C05463=1023.749,201.807,381.412,168.832,48.309,159.110
C05464=1023.754,202.056,381.388,168.836,48.304,159.109
C05465=1023.760,202.305,381.365,168.841,48.300,159.109
C05466=1023.765,202.553,381.340,168.844,48.295,159.109
C05467=1023.771,202.803,381.316,168.849,48.290,159.108
C05468=1023.776,203.051,381.291,168.853,48.285,159.108
C05469=1023.782,203.300,381.268,168.857,48.280,159.107
C05470=1023.805,204.331,381.167,169.270,48.380,159.187
C05471=1023.816,204.745,381.124,169.275,48.373,159.186
C05472=1023.827,205.160,381.081,169.281,48.366,159.186
C05473=1023.838,205.574,381.039,169.286,48.359,159.185
C05474=1023.849,205.988,380.996,169.292,48.352,159.184
C05475=1023.856,206.237,380.969,169.295,48.349,159.184
C05476=1023.862,206.486,380.944,169.298,48.344,159.184
C05477=1023.868,206.734,380.918,169.301,48.341,159.183
C05478=1023.874,206.982,380.892,169.305,48.336,159.183
C05479=1023.882,207.231,380.866,169.307,48.333,159.182
C05480=1023.888,207.480,380.841,169.311,48.329,159.182
C05481=1023.894,207.728,380.815,169.314,48.325,159.182
C05482=1023.900,207.976,380.789,169.318,48.321,159.181
C05483=1023.908,208.225,380.763,169.320,48.317,159.181
C05484=1023.913,208.474,380.737,169.324,48.313,159.180
C05485=1023.920,208.722,380.711,169.327,48.309,159.180
C05486=1023.926,208.972,380.685,169.331,48.305,159.180
C05487=1023.933,209.220,380.659,169.333,48.301,159.179
C05488=1023.939,209.468,380.633,169.337,48.297,159.179
C05489=1023.946,209.717,380.607,169.340,48.293,159.179
C05490=1023.952,209.965,380.581,169.344,48.289,159.178
C05491=1023.958,210.214,380.555,169.346,48.285,159.178
C05492=1023.965,210.462,380.529,169.350,48.282,159.178
C05493=1023.972,210.711,380.503,169.353,48.278,159.177
C05494=1023.978,210.959,380.476,169.356,48.274,159.177
C05495=1023.984,211.208,380.451,169.360,48.270,159.176
C05496=1023.991,211.457,380.425,169.362,48.266,159.176
C05497=1023.997,211.705,380.398,169.366,48.263,159.176
C05498=1024.003,211.954,380.373,169.369,48.259,159.175
C05499=1024.009,212.203,380.346,169.373,48.255,159.175
C05500=1024.016,212.451,380.319,169.376,48.251,159.175
C05501=1024.022,212.699,380.293,169.379,48.247,159.174
C05502=1024.029,212.948,380.266,169.382,48.244,159.174
C05503=1024.035,213.197,380.241,169.386,48.240,159.174
C05504=1024.042,213.445,380.215,169.389,48.236,159.173
C05505=1024.048,213.694,380.188,169.393,48.232,159.173
C05506=1024.054,213.942,380.162,169.396,48.229,159.173
C05507=1024.061,214.191,380.135,169.399,48.225,159.172
C05508=1024.067,214.439,380.110,169.402,48.221,159.172
C05509=1024.073,214.688,380.084,169.406,48.217,159.172
C05510=1024.080,214.937,380.057,169.409,48.214,159.171
C05511=1024.086,215.185,380.030,169.412,48.210,159.171
C05512=1024.093,215.433,380.004,169.415,48.206,159.171
C05513=1024.099,215.682,379.977,169.418,48.202,159.170
C05514=1024.106,215.930,379.951,169.422,48.198,159.170
C05515=1024.112,216.179,379.924,169.425,48.195,159.170
C05516=1024.119,216.427,379.898,169.429,48.191,159.169
C05517=1024.125,216.676,379.873,169.432,48.187,159.169
C05518=1024.131,216.925,379.846,169.435,48.183,159.169
C05519=1024.138,217.173,379.819,169.439,48.180,159.168
C05520=1024.145,217.421,379.793,169.442,48.176,159.168
C05521=1024.151,217.670,379.766,169.445,48.172,159.168
C05522=1024.158,217.919,379.740,169.449,48.169,159.167
C05523=1024.164,218.168,379.713,169.452,48.165,159.167
C05524=1024.171,218.416,379.687,169.456,48.161,159.167
C05525=1024.178,218.664,379.661,169.459,48.158,159.166
C05526=1024.183,218.913,379.634,169.462,48.154,159.166
C05527=1024.194,219.329,379.590,169.468,48.148,159.165
C05528=1024.205,219.746,379.544,169.474,48.142,159.165
C05529=1024.215,220.162,379.500,169.479,48.136,159.165
C05530=1024.227,220.579,379.455,169.485,48.130,159.164
C05531=1024.232,220.828,379.428,169.488,48.127,159.164
C05532=1024.239,221.077,379.401,169.491,48.123,159.163
C05533=1024.245,221.325,379.375,169.495,48.120,159.163
C05534=1024.252,221.574,379.348,169.498,48.116,159.163
C05535=1024.258,221.822,379.321,169.502,48.112,159.163
C05536=1024.265,222.070,379.294,169.505,48.109,159.162
C05537=1024.271,222.319,379.268,169.509,48.105,159.162
C05538=1024.277,222.568,379.241,169.512,48.102,159.162
C05539=1024.284,222.815,379.214,169.516,48.098,159.161
C05540=1024.290,223.064,379.187,169.519,48.095,159.161
C05541=1024.297,223.313,379.160,169.521,48.091,159.161
C05542=1024.303,223.561,379.134,169.525,48.088,159.161
C05543=1024.310,223.810,379.106,169.529,48.085,159.160
C05544=1024.316,224.058,379.079,169.532,48.080,159.160
C05545=1024.323,224.307,379.053,169.535,48.077,159.160
C05546=1024.329,224.555,379.025,169.539,48.074,159.160
C05547=1024.335,224.804,378.998,169.542,48.070,159.159
C05548=1024.342,225.053,378.972,169.546,48.067,159.159
C05549=1024.348,225.300,378.945,169.549,48.064,159.159
C05550=1024.355,225.549,378.918,169.553,48.060,159.158
C05551=1024.361,225.797,378.892,169.556,48.056,159.158
C05552=1024.368,226.046,378.864,169.560,48.053,159.158
C05553=1024.374,226.295,378.837,169.563,48.049,159.158
C05554=1024.380,226.543,378.810,169.567,48.046,159.157
C05555=1024.388,226.791,378.783,169.570,48.043,159.157
C05556=1024.394,227.040,378.756,169.573,48.039,159.157
C05557=1024.400,227.288,378.729,169.577,48.035,159.157
C05558=1024.406,227.537,378.702,169.580,48.032,159.156
C05559=1024.412,227.785,378.674,169.584,48.029,159.156
C05560=1024.420,228.034,378.648,169.587,48.026,159.156
C05561=1024.426,228.282,378.620,169.591,48.022,159.156
C05562=1024.432,228.531,378.594,169.594,48.019,159.155
C05563=1024.439,228.779,378.566,169.598,48.015,159.155
C05564=1024.445,229.028,378.539,169.601,48.012,159.155
C05565=1024.451,229.276,378.511,169.604,48.009,159.155
C05566=1024.458,229.524,378.484,169.608,48.006,159.154
C05567=1024.464,229.773,378.457,169.611,48.003,159.154
C05568=1024.470,230.021,378.429,169.616,47.999,159.154
C05569=1024.477,230.269,378.402,169.618,47.995,159.154
C05570=1024.483,230.519,378.375,169.622,47.992,159.153
C05571=1024.490,230.767,378.347,169.625,47.989,159.153
C05572=1024.496,231.015,378.319,169.629,47.986,159.153
C05573=1024.502,231.264,378.292,169.633,47.982,159.153
C05574=1024.509,231.512,378.265,169.636,47.979,159.153
C05575=1024.515,231.760,378.237,169.640,47.976,159.152
C05576=1024.522,232.009,378.210,169.643,47.973,159.152
C05577=1024.528,232.257,378.183,169.647,47.969,159.152
C05578=1024.534,232.505,378.155,169.650,47.966,159.152
C05579=1024.541,232.754,378.128,169.653,47.963,159.151
C05580=1024.548,233.002,378.100,169.657,47.960,159.151
C05581=1024.553,233.251,378.072,169.660,47.957,159.151
C05582=1024.559,233.499,378.045,169.664,47.953,159.151
C05583=1024.570,233.908,378.000,169.670,47.949,159.151
C05584=1024.581,234.317,377.955,169.676,47.943,159.150
C05585=1024.591,234.726,377.908,169.682,47.938,159.150
C05586=1024.602,235.134,377.863,169.688,47.932,159.150
C05587=1024.609,235.383,377.835,169.691,47.929,159.149
C05588=1024.615,235.631,377.808,169.695,47.926,159.149
C05589=1024.622,235.880,377.781,169.698,47.923,159.149
C05590=1024.628,236.129,377.753,169.702,47.919,159.149
C05591=1024.634,236.377,377.726,169.705,47.917,159.149
C05592=1024.641,236.625,377.698,169.709,47.914,159.148
C05593=1024.647,236.874,377.669,169.712,47.910,159.148
C05594=1024.654,237.122,377.642,169.717,47.907,159.148
C05595=1024.660,237.371,377.614,169.720,47.904,159.148
C05596=1024.667,237.619,377.586,169.723,47.901,159.147
C05597=1024.673,237.867,377.559,169.727,47.898,159.148
C05598=1024.680,238.115,377.531,169.730,47.895,159.147
C05599=1024.686,238.364,377.503,169.734,47.892,159.147
C05600=1024.693,238.612,377.475,169.737,47.888,159.147
C05601=1024.699,238.861,377.447,169.741,47.885,159.147
C05602=1024.706,239.109,377.420,169.745,47.883,159.147
C05603=1024.713,239.358,377.392,169.749,47.879,159.146
C05604=1024.719,239.606,377.364,169.752,47.876,159.146
C05605=1024.725,239.854,377.336,169.755,47.873,159.146
C05606=1024.732,240.102,377.308,169.759,47.870,159.146
C05607=1024.738,240.351,377.280,169.763,47.867,159.146
C05608=1024.744,240.599,377.252,169.767,47.864,159.145
C05609=1024.751,240.848,377.224,169.770,47.861,159.145
C05610=1024.757,241.096,377.195,169.774,47.858,159.145
C05611=1024.764,241.344,377.167,169.777,47.855,159.145
C05612=1024.770,241.593,377.139,169.781,47.852,159.145
C05613=1024.776,241.841,377.112,169.785,47.849,159.145
C05614=1024.783,242.089,377.083,169.788,47.847,159.145
C05615=1024.789,242.337,377.055,169.792,47.843,159.144
C05616=1024.795,242.586,377.027,169.795,47.840,159.144
C05617=1024.802,242.834,376.998,169.800,47.837,159.144
C05618=1024.808,243.082,376.970,169.803,47.834,159.144
C05619=1024.814,243.331,376.942,169.806,47.832,159.144
C05620=1024.821,243.579,376.914,169.810,47.829,159.144
C05621=1024.828,243.827,376.886,169.814,47.826,159.144
C05622=1024.834,244.076,376.857,169.818,47.823,159.143
C05623=1024.840,244.324,376.828,169.821,47.820,159.143
C05624=1024.847,244.573,376.801,169.824,47.817,159.143
C05625=1024.853,244.821,376.772,169.829,47.814,159.143
C05626=1024.859,245.070,376.743,169.832,47.812,159.143
C05627=1024.865,245.317,376.715,169.836,47.809,159.143
C05628=1024.871,245.565,376.687,169.840,47.806,159.143
C05629=1024.878,245.814,376.658,169.843,47.803,159.143
C05630=1024.884,246.062,376.629,169.847,47.800,159.143
C05631=1024.891,246.310,376.601,169.850,47.798,159.143
C05632=1024.897,246.558,376.572,169.855,47.795,159.142
C05633=1024.903,246.807,376.544,169.858,47.792,159.142
C05634=1024.909,247.055,376.515,169.861,47.790,159.142
C05635=1024.916,247.304,376.487,169.865,47.786,159.142
C05636=1024.922,247.552,376.458,169.869,47.784,159.142
C05637=1024.928,247.800,376.429,169.873,47.781,159.142
C05638=1024.935,248.048,376.401,169.876,47.778,159.142
C05639=1024.945,248.451,376.355,169.882,47.773,159.141
C05640=1024.955,248.854,376.307,169.888,47.769,159.141
C05641=1024.966,249.256,376.261,169.895,47.765,159.141
C05642=1024.976,249.660,376.215,169.901,47.760,159.141
C05643=1024.983,249.908,376.186,169.904,47.758,159.141
C05644=1024.990,250.156,376.157,169.909,47.755,159.141
C05645=1024.996,250.404,376.128,169.912,47.752,159.141
C05646=1025.002,250.652,376.100,169.916,47.749,159.141
C05647=1025.009,250.900,376.072,169.920,47.747,159.141
C05648=1025.015,251.148,376.042,169.923,47.744,159.141
C05649=1025.021,251.397,376.013,169.927,47.741,159.141
C05650=1025.027,251.645,375.985,169.931,47.738,159.140
C05651=1025.035,251.894,375.956,169.935,47.736,159.140
C05652=1025.041,252.142,375.927,169.938,47.733,159.140
C05653=1025.047,252.390,375.898,169.943,47.731,159.140
C05654=1025.053,252.638,375.869,169.946,47.728,159.140
C05655=1025.060,252.887,375.841,169.950,47.725,159.140
C05656=1025.066,253.135,375.812,169.954,47.722,159.140
C05657=1025.073,253.383,375.783,169.958,47.720,159.140
C05658=1025.080,253.631,375.755,169.962,47.717,159.140
C05659=1025.086,253.880,375.726,169.965,47.715,159.140
C05660=1025.093,254.128,375.696,169.969,47.712,159.140
C05661=1025.099,254.376,375.667,169.972,47.709,159.139
C05662=1025.106,254.624,375.639,169.977,47.706,159.139
C05663=1025.113,254.872,375.610,169.980,47.704,159.139
C05664=1025.119,255.121,375.581,169.985,47.701,159.139
C05665=1025.125,255.369,375.552,169.988,47.699,159.139
C05666=1025.132,255.617,375.524,169.992,47.696,159.139
C05667=1025.139,255.866,375.494,169.996,47.693,159.139
C05668=1025.145,256.114,375.465,170.000,47.691,159.139
C05669=1025.151,256.362,375.436,170.003,47.688,159.139
C05670=1025.158,256.610,375.408,170.008,47.685,159.139
C05671=1025.165,256.859,375.378,170.011,47.683,159.139
C05672=1025.171,257.107,375.349,170.016,47.680,159.139
C05673=1025.178,257.355,375.320,170.019,47.677,159.139
C05674=1025.186,257.603,375.291,170.023,47.675,159.139
C05675=1025.192,257.851,375.262,170.027,47.672,159.139
C05676=1025.198,258.099,375.233,170.031,47.670,159.139
C05677=1025.204,258.347,375.204,170.035,47.667,159.139
C05678=1025.212,258.596,375.175,170.039,47.664,159.139
C05679=1025.218,258.844,375.146,170.043,47.662,159.139
C05680=1025.224,259.092,375.117,170.047,47.659,159.139
C05681=1025.231,259.341,375.087,170.050,47.657,159.138
C05682=1025.238,259.589,375.059,170.055,47.654,159.138
C05683=1025.245,259.838,375.030,170.058,47.652,159.138
C05684=1025.252,260.085,375.000,170.063,47.649,159.138
C05685=1025.258,260.333,374.971,170.066,47.647,159.138
C05686=1025.266,260.582,374.942,170.070,47.644,159.138
C05687=1025.272,260.830,374.913,170.074,47.641,159.138
C05688=1025.278,261.078,374.883,170.079,47.639,159.138
C05689=1025.284,261.327,374.853,170.082,47.637,159.138
C05690=1025.291,261.575,374.824,170.086,47.634,159.138
C05691=1025.297,261.822,374.794,170.090,47.632,159.138
C05692=1025.304,262.071,374.765,170.094,47.629,159.138
C05693=1025.311,262.319,374.735,170.098,47.627,159.138
C05694=1025.317,262.567,374.706,170.102,47.625,159.138
C05695=1025.327,262.968,374.657,170.108,47.621,159.138
C05696=1025.338,263.369,374.610,170.115,47.617,159.138
C05697=1025.348,263.771,374.562,170.121,47.614,159.138
C05698=1025.359,264.172,374.514,170.128,47.609,159.138
C05699=1025.365,264.420,374.484,170.132,47.607,159.138
C05700=1025.372,264.668,374.455,170.136,47.605,159.138
C05701=1025.379,264.916,374.425,170.140,47.602,159.138
C05702=1025.384,265.164,374.396,170.143,47.600,159.138
C05703=1025.391,265.413,374.366,170.148,47.598,159.138
C05704=1025.398,265.660,374.336,170.151,47.596,159.138
C05705=1025.405,265.909,374.306,170.156,47.593,159.138
C05706=1025.411,266.156,374.277,170.159,47.591,159.138
C05707=1025.418,266.405,374.246,170.164,47.588,159.138
C05708=1025.424,266.653,374.217,170.168,47.587,159.139
C05709=1025.431,266.901,374.187,170.172,47.584,159.139
C05710=1025.437,267.149,374.156,170.176,47.582,159.139
C05711=1025.444,267.398,374.127,170.180,47.579,159.139
C05712=1025.450,267.645,374.097,170.184,47.578,159.139
C05713=1025.458,267.894,374.067,170.188,47.575,159.139
C05714=1025.463,268.141,374.037,170.192,47.573,159.139
C05715=1025.470,268.390,374.007,170.196,47.571,159.139
C05716=1025.476,268.638,373.977,170.200,47.569,159.139
C05717=1025.483,268.886,373.947,170.205,47.566,159.139
C05718=1025.490,269.134,373.917,170.208,47.564,159.139
C05719=1025.496,269.382,373.886,170.213,47.562,159.139
C05720=1025.503,269.630,373.857,170.216,47.560,159.139
C05721=1025.510,269.879,373.827,170.221,47.557,159.139
C05722=1025.515,270.126,373.797,170.225,47.555,159.139
C05723=1025.523,270.375,373.767,170.229,47.553,159.139
C05724=1025.528,270.623,373.736,170.233,47.551,159.139
C05725=1025.536,270.871,373.706,170.237,47.549,159.139
C05726=1025.541,271.119,373.676,170.241,47.546,159.139
C05727=1025.549,271.367,373.646,170.246,47.544,159.140
C05728=1025.555,271.615,373.615,170.249,47.543,159.140
C05729=1025.562,271.863,373.585,170.254,47.540,159.140
C05730=1025.568,272.111,373.555,170.257,47.538,159.140
C05731=1025.575,272.359,373.525,170.262,47.536,159.140
C05732=1025.581,272.607,373.494,170.266,47.534,159.140
C05733=1025.588,272.856,373.464,170.270,47.532,159.140
C05734=1025.594,273.103,373.434,170.274,47.530,159.140
C05735=1025.601,273.352,373.404,170.279,47.528,159.140
C05736=1025.607,273.599,373.372,170.282,47.526,159.140
C05737=1025.614,273.847,373.342,170.287,47.523,159.140
C05738=1025.621,274.096,373.312,170.292,47.521,159.140
C05739=1025.627,274.343,373.282,170.295,47.520,159.141
C05740=1025.634,274.592,373.251,170.300,47.517,159.141
C05741=1025.640,274.840,373.220,170.304,47.516,159.141
C05742=1025.647,275.087,373.190,170.308,47.513,159.141
C05743=1025.653,275.336,373.159,170.312,47.511,159.141
C05744=1025.661,275.584,373.129,170.317,47.509,159.141
C05745=1025.666,275.832,373.099,170.320,47.507,159.141
C05746=1025.673,276.079,373.067,170.325,47.505,159.141
C05747=1025.680,276.328,373.037,170.329,47.504,159.141
C05748=1025.687,276.576,373.007,170.333,47.501,159.141
C05749=1025.693,276.824,372.977,170.337,47.499,159.142
C05750=1025.700,277.072,372.945,170.342,47.497,159.142
C05751=1025.711,277.478,372.895,170.348,47.494,159.142
C05752=1025.721,277.883,372.845,170.356,47.491,159.142
C05753=1025.732,278.289,372.795,170.362,47.488,159.142
C05754=1025.743,278.695,372.743,170.370,47.485,159.143
C05755=1025.749,278.943,372.713,170.374,47.483,159.143
C05756=1025.756,279.190,372.682,170.379,47.481,159.143
C05757=1025.762,279.439,372.652,170.382,47.479,159.143
C05758=1025.769,279.687,372.620,170.387,47.477,159.143
C05759=1025.776,279.935,372.589,170.391,47.475,159.143
C05760=1025.782,280.182,372.558,170.395,47.473,159.143
C05761=1025.788,280.431,372.528,170.399,47.472,159.144
C05762=1025.795,280.679,372.496,170.404,47.470,159.144
C05763=1025.802,280.926,372.465,170.408,47.468,159.144
C05764=1025.809,281.175,372.435,170.413,47.466,159.144
C05765=1025.815,281.422,372.404,170.417,47.464,159.144
C05766=1025.821,281.671,372.373,170.421,47.463,159.144
C05767=1025.828,281.919,372.341,170.426,47.461,159.145
C05768=1025.835,282.167,372.310,170.430,47.459,159.145
C05769=1025.842,282.415,372.280,170.434,47.457,159.145
C05770=1025.849,282.663,372.248,170.438,47.455,159.145
C05771=1025.855,282.911,372.217,170.443,47.454,159.145
C05772=1025.861,283.158,372.186,170.448,47.452,159.145
C05773=1025.868,283.406,372.155,170.452,47.450,159.146
C05774=1025.875,283.654,372.124,170.456,47.448,159.146
C05775=1025.881,283.902,372.092,170.460,47.447,159.146
C05776=1025.889,284.150,372.062,170.465,47.445,159.146
C05777=1025.895,284.398,372.031,170.469,47.443,159.146
C05778=1025.902,284.646,371.999,170.474,47.441,159.146
C05779=1025.909,284.894,371.968,170.478,47.439,159.147
C05780=1025.915,285.142,371.936,170.482,47.438,159.147
C05781=1025.922,285.390,371.905,170.487,47.436,159.147
C05782=1025.929,285.638,371.874,170.491,47.434,159.147
C05783=1025.935,285.886,371.843,170.496,47.432,159.147
C05784=1025.941,286.133,371.812,170.501,47.430,159.148
C05785=1025.948,286.381,371.780,170.505,47.429,159.148
C05786=1025.955,286.629,371.749,170.509,47.427,159.148
C05787=1025.962,286.877,371.718,170.513,47.426,159.148
C05788=1025.968,287.125,371.686,170.518,47.424,159.148
C05789=1025.975,287.373,371.655,170.523,47.422,159.149
C05790=1025.982,287.621,371.623,170.527,47.421,159.149
C05791=1025.989,287.868,371.591,170.532,47.419,159.149
C05792=1025.995,288.116,371.560,170.536,47.418,159.149
C05793=1026.001,288.364,371.528,170.540,47.416,159.150
C05794=1026.008,288.612,371.496,170.545,47.414,159.150
C05795=1026.015,288.860,371.465,170.549,47.413,159.150
C05796=1026.022,289.108,371.433,170.554,47.411,159.150
C05797=1026.028,289.356,371.402,170.558,47.409,159.150
C05798=1026.035,289.603,371.370,170.563,47.408,159.151
C05799=1026.043,289.852,371.338,170.568,47.406,159.151
C05800=1026.049,290.100,371.306,170.572,47.405,159.151
C05801=1026.055,290.348,371.275,170.576,47.403,159.151
C05802=1026.062,290.596,371.243,170.581,47.401,159.152
C05803=1026.069,290.843,371.211,170.586,47.400,159.152
C05804=1026.076,291.091,371.179,170.590,47.398,159.152
C05805=1026.082,291.339,371.147,170.594,47.397,159.152
C05806=1026.089,291.586,371.115,170.599,47.395,159.153
C05807=1026.101,292.005,371.062,170.607,47.393,159.153
C05808=1026.112,292.423,371.008,170.615,47.390,159.153
C05809=1026.123,292.840,370.954,170.623,47.388,159.154
C05810=1026.134,293.259,370.901,170.630,47.385,159.154
C05811=1026.141,293.506,370.869,170.635,47.384,159.155
C05812=1026.148,293.755,370.836,170.640,47.382,159.155
C05813=1026.155,294.002,370.804,170.644,47.381,159.155
C05814=1026.161,294.250,370.772,170.649,47.379,159.155
C05815=1026.168,294.498,370.740,170.654,47.378,159.156
C05816=1026.174,294.745,370.707,170.658,47.377,159.156
C05817=1026.180,294.993,370.675,170.663,47.375,159.156
C05818=1026.187,295.241,370.643,170.667,47.374,159.157
C05819=1026.194,295.489,370.610,170.672,47.373,159.157
C05820=1026.201,295.736,370.578,170.677,47.371,159.157
C05821=1026.207,295.985,370.546,170.681,47.370,159.158
C05822=1026.213,296.232,370.513,170.686,47.369,159.158
C05823=1026.221,296.479,370.481,170.690,47.368,159.158
C05824=1026.227,296.728,370.448,170.695,47.366,159.158
C05825=1026.233,296.976,370.416,170.700,47.365,159.159
C05826=1026.240,297.223,370.384,170.704,47.364,159.159
C05827=1026.247,297.471,370.351,170.709,47.362,159.159
C05828=1026.253,297.718,370.318,170.714,47.361,159.160
C05829=1026.261,297.966,370.286,170.718,47.360,159.160
C05830=1026.267,298.215,370.254,170.723,47.358,159.160
C05831=1026.273,298.462,370.221,170.728,47.357,159.161
C05832=1026.280,298.709,370.189,170.732,47.356,159.161
C05833=1026.287,298.958,370.156,170.737,47.355,159.161
C05834=1026.294,299.205,370.124,170.742,47.353,159.162
C05835=1026.300,299.453,370.091,170.747,47.353,159.162
C05836=1026.307,299.701,370.058,170.752,47.351,159.162
C05837=1026.314,299.948,370.026,170.757,47.350,159.163
C05838=1026.320,300.196,369.993,170.761,47.349,159.163
C05839=1026.327,300.444,369.960,170.766,47.347,159.163
C05840=1026.334,300.691,369.928,170.771,47.346,159.164
C05841=1026.341,300.939,369.895,170.775,47.345,159.164
C05842=1026.347,301.187,369.862,170.780,47.344,159.165
C05843=1026.355,301.435,369.830,170.785,47.343,159.165
C05844=1026.361,301.683,369.796,170.790,47.341,159.165
C05845=1026.368,301.930,369.764,170.794,47.340,159.165
C05846=1026.375,302.178,369.732,170.799,47.339,159.166
C05847=1026.382,302.426,369.698,170.805,47.338,159.166
C05848=1026.388,302.673,369.665,170.810,47.337,159.167
C05849=1026.396,302.921,369.632,170.814,47.335,159.167
C05850=1026.402,303.169,369.600,170.819,47.334,159.167
C05851=1026.408,303.416,369.567,170.824,47.333,159.168
C05852=1026.416,303.664,369.534,170.828,47.332,159.168
C05853=1026.422,303.912,369.502,170.833,47.331,159.168
C05854=1026.430,304.159,369.468,170.839,47.330,159.169
C05855=1026.437,304.407,369.436,170.844,47.329,159.169
C05856=1026.444,304.655,369.403,170.848,47.328,159.169
C05857=1026.450,304.903,369.370,170.853,47.327,159.170
C05858=1026.458,305.150,369.337,170.858,47.325,159.170
C05859=1026.464,305.397,369.304,170.863,47.324,159.171
C05860=1026.471,305.646,369.271,170.869,47.323,159.171
C05861=1026.479,305.893,369.238,170.873,47.322,159.171
C05862=1026.485,306.141,369.205,170.878,47.321,159.172
C05863=1026.491,306.358,369.176,170.882,47.320,159.172
C05864=1026.497,306.576,369.147,170.887,47.319,159.173
C05865=1026.504,306.794,369.118,170.891,47.318,159.173
C05866=1026.510,307.012,369.089,170.895,47.317,159.173
C05867=1026.516,307.228,369.059,170.899,47.316,159.174
C05868=1026.522,307.446,369.030,170.904,47.316,159.174
C05869=1026.529,307.664,369.001,170.909,47.314,159.174
C05870=1026.534,307.882,368.972,170.913,47.313,159.175
C05871=1026.542,308.130,368.940,170.918,47.312,159.175
C05872=1026.548,308.377,368.906,170.923,47.311,159.175
C05873=1026.555,308.625,368.873,170.928,47.310,159.176
C05874=1026.563,308.873,368.840,170.933,47.309,159.176
C05875=1026.570,309.120,368.806,170.938,47.308,159.177
C05876=1026.577,309.368,368.773,170.943,47.307,159.177
C05877=1026.584,309.616,368.739,170.948,47.306,159.178
C05878=1026.591,309.863,368.707,170.954,47.305,159.178
C05879=1026.598,310.110,368.673,170.958,47.304,159.178
C05880=1026.605,310.358,368.640,170.963,47.303,159.179
C05881=1026.612,310.605,368.607,170.968,47.302,159.179
C05882=1026.620,310.853,368.574,170.973,47.301,159.180
C05883=1026.626,311.101,368.539,170.979,47.300,159.180
C05884=1026.633,311.348,368.506,170.983,47.300,159.181
C05885=1026.640,311.596,368.472,170.989,47.299,159.181
C05886=1026.647,311.843,368.438,170.994,47.298,159.182
C05887=1026.653,312.091,368.404,170.999,47.297,159.182
C05888=1026.660,312.338,368.370,171.004,47.296,159.183
C05889=1026.667,312.586,368.336,171.009,47.296,159.183
C05890=1026.674,312.834,368.302,171.014,47.295,159.184
C05891=1026.680,313.081,368.268,171.019,47.294,159.184
C05892=1026.688,313.329,368.235,171.025,47.293,159.185
C05893=1026.694,313.577,368.200,171.030,47.293,159.185
C05894=1026.701,313.824,368.167,171.034,47.292,159.186
C05895=1026.708,314.071,368.133,171.040,47.291,159.186
C05896=1026.714,314.319,368.099,171.045,47.291,159.187
C05897=1026.721,314.567,368.065,171.050,47.290,159.187
C05898=1026.729,314.815,368.031,171.056,47.289,159.188
C05899=1026.735,315.062,367.997,171.061,47.288,159.188
C05900=1026.742,315.309,367.962,171.065,47.288,159.189
C05901=1026.749,315.557,367.928,171.071,47.287,159.189
C05902=1026.756,315.805,367.894,171.076,47.286,159.190
C05903=1026.763,316.052,367.860,171.082,47.286,159.190
C05904=1026.770,316.300,367.826,171.087,47.285,159.191
C05905=1026.776,316.547,367.792,171.092,47.284,159.191
C05906=1026.783,316.794,367.758,171.098,47.283,159.192
C05907=1026.791,317.042,367.724,171.102,47.283,159.192
C05908=1026.797,317.290,367.690,171.108,47.283,159.193
C05909=1026.805,317.537,367.655,171.113,47.282,159.193
C05910=1026.812,317.785,367.621,171.118,47.281,159.194
C05911=1026.818,318.033,367.587,171.124,47.280,159.194
C05912=1026.826,318.280,367.552,171.129,47.280,159.195
C05913=1026.833,318.527,367.518,171.134,47.279,159.195
C05914=1026.840,318.775,367.483,171.140,47.279,159.196
C05915=1026.847,319.022,367.449,171.145,47.278,159.197
C05916=1026.854,319.270,367.416,171.150,47.277,159.197
C05917=1026.861,319.517,367.381,171.155,47.277,159.198
C05918=1026.868,319.765,367.347,171.161,47.276,159.198
C05919=1026.876,320.012,367.312,171.166,47.276,159.199
C05920=1026.882,320.260,367.278,171.171,47.275,159.199
C05921=1026.890,320.507,367.243,171.177,47.274,159.200
C05922=1026.897,320.755,367.209,171.182,47.274,159.200
C05923=1026.903,320.975,367.178,171.187,47.273,159.201
C05924=1026.909,321.196,367.147,171.192,47.273,159.201
C05925=1026.915,321.415,367.116,171.196,47.272,159.202
C05926=1026.922,321.636,367.086,171.202,47.272,159.203
C05927=1026.928,321.856,367.055,171.206,47.272,159.203
C05928=1026.935,322.076,367.024,171.212,47.271,159.203
C05929=1026.941,322.296,366.994,171.216,47.270,159.204
C05930=1026.948,322.516,366.963,171.220,47.270,159.204
C05931=1026.955,322.763,366.929,171.226,47.270,159.205
C05932=1026.962,323.011,366.894,171.231,47.269,159.206
C05933=1026.970,323.258,366.859,171.237,47.269,159.206
C05934=1026.977,323.506,366.825,171.242,47.268,159.207
C05935=1026.984,323.754,366.790,171.248,47.268,159.207
C05936=1026.991,324.001,366.756,171.253,47.267,159.208
C05937=1026.999,324.248,366.721,171.259,47.267,159.209
C05938=1027.006,324.496,366.686,171.265,47.266,159.209
C05939=1027.013,324.743,366.652,171.270,47.266,159.210
C05940=1027.020,324.991,366.617,171.276,47.265,159.210
C05941=1027.028,325.239,366.582,171.281,47.265,159.211
C05942=1027.036,325.486,366.547,171.287,47.264,159.212
C05943=1027.042,325.733,366.512,171.293,47.264,159.212
C05944=1027.050,325.981,366.478,171.299,47.263,159.213
C05945=1027.057,326.229,366.443,171.304,47.263,159.214
C05946=1027.064,326.476,366.408,171.310,47.263,159.214
C05947=1027.073,326.723,366.373,171.315,47.262,159.215
C05948=1027.079,326.971,366.338,171.321,47.262,159.215
C05949=1027.087,327.218,366.304,171.327,47.262,159.216
C05950=1027.094,327.466,366.268,171.332,47.261,159.217
C05951=1027.102,327.713,366.234,171.338,47.261,159.217
C05952=1027.109,327.960,366.198,171.343,47.261,159.218
C05953=1027.116,328.208,366.162,171.349,47.260,159.219
C05954=1027.123,328.455,366.127,171.355,47.260,159.219
C05955=1027.130,328.703,366.092,171.360,47.259,159.220
C05956=1027.138,328.950,366.056,171.366,47.259,159.221
C05957=1027.145,329.197,366.021,171.371,47.259,159.221
C05958=1027.152,329.444,365.986,171.377,47.259,159.222
C05959=1027.159,329.692,365.950,171.382,47.259,159.223
C05960=1027.166,329.939,365.915,171.388,47.259,159.223
C05961=1027.173,330.187,365.879,171.394,47.259,159.224
C05962=1027.181,330.434,365.844,171.400,47.258,159.225
C05963=1027.188,330.681,365.809,171.406,47.258,159.226
C05964=1027.195,330.929,365.773,171.412,47.258,159.226
C05965=1027.202,331.176,365.737,171.417,47.258,159.227
C05966=1027.210,331.424,365.702,171.423,47.257,159.228
C05967=1027.217,331.671,365.666,171.429,47.257,159.228
C05968=1027.225,331.918,365.631,171.434,47.257,159.229
C05969=1027.232,332.165,365.595,171.440,47.257,159.230
C05970=1027.239,332.413,365.560,171.446,47.257,159.230
C05971=1027.247,332.660,365.524,171.451,47.257,159.231
C05972=1027.254,332.908,365.488,171.458,47.256,159.232
C05973=1027.262,333.156,365.452,171.464,47.257,159.233
C05974=1027.269,333.402,365.417,171.470,47.257,159.233
C05975=1027.277,333.650,365.381,171.475,47.256,159.234
C05976=1027.284,333.897,365.346,171.481,47.256,159.235
C05977=1027.292,334.144,365.309,171.487,47.256,159.236
C05978=1027.298,334.392,365.274,171.493,47.256,159.236
C05979=1027.306,334.639,365.238,171.499,47.256,159.237
C05980=1027.313,334.887,365.201,171.505,47.256,159.238
C05981=1027.320,335.134,365.165,171.511,47.256,159.239
C05982=1027.328,335.381,365.129,171.517,47.256,159.239
C05983=1027.334,335.598,365.098,171.521,47.256,159.240
C05984=1027.340,335.817,365.066,171.527,47.256,159.241
C05985=1027.348,336.035,365.034,171.533,47.256,159.241
C05986=1027.354,336.252,365.003,171.537,47.256,159.242
C05987=1027.360,336.470,364.971,171.543,47.256,159.243
C05988=1027.367,336.688,364.939,171.548,47.257,159.244
C05989=1027.373,336.906,364.907,171.553,47.256,159.244
C05990=1027.380,337.124,364.875,171.558,47.257,159.245
C05991=1027.387,337.372,364.839,171.565,47.256,159.246
C05992=1027.394,337.618,364.803,171.571,47.257,159.247
C05993=1027.402,337.866,364.767,171.576,47.256,159.247
C05994=1027.410,338.113,364.731,171.582,47.257,159.248
C05995=1027.417,338.361,364.694,171.588,47.257,159.249
C05996=1027.424,338.608,364.658,171.595,47.257,159.250
C05997=1027.432,338.855,364.622,171.601,47.257,159.250
C05998=1027.439,339.102,364.585,171.607,47.257,159.251
C05999=1027.447,339.349,364.549,171.613,47.258,159.252
C06000=1027.455,339.597,364.512,171.619,47.257,159.253
C06001=1027.462,339.844,364.477,171.625,47.258,159.254
C06002=1027.470,340.091,364.440,171.631,47.258,159.255
C06003=1027.478,340.338,364.403,171.637,47.258,159.255
C06004=1027.485,340.586,364.367,171.644,47.258,159.256
C06005=1027.492,340.833,364.330,171.650,47.258,159.257
C06006=1027.500,341.080,364.293,171.655,47.258,159.258
C06007=1027.507,341.328,364.257,171.661,47.259,159.259
C06008=1027.514,341.574,364.220,171.668,47.259,159.260
C06009=1027.522,341.821,364.184,171.674,47.259,159.261
C06010=1027.529,342.068,364.146,171.680,47.260,159.261
C06011=1027.537,342.316,364.110,171.686,47.260,159.262
C06012=1027.544,342.563,364.073,171.693,47.260,159.263
C06013=1027.552,342.810,364.036,171.699,47.260,159.264
C06014=1027.560,343.057,363.999,171.705,47.261,159.265
C06015=1027.567,343.305,363.963,171.712,47.261,159.266
C06016=1027.575,343.552,363.926,171.718,47.261,159.267
C06017=1027.583,343.799,363.889,171.724,47.262,159.268
C06018=1027.590,344.046,363.852,171.731,47.262,159.268
C06019=1027.598,344.293,363.815,171.737,47.262,159.269
C06020=1027.605,344.540,363.777,171.743,47.263,159.270
C06021=1027.613,344.788,363.741,171.750,47.263,159.271
C06022=1027.620,345.035,363.704,171.756,47.263,159.272
C06023=1027.628,345.282,363.667,171.762,47.264,159.273
C06024=1027.635,345.529,363.629,171.769,47.264,159.274
C06025=1027.643,345.776,363.593,171.775,47.264,159.275
C06026=1027.651,346.023,363.556,171.781,47.265,159.276
C06027=1027.658,346.270,363.519,171.788,47.266,159.277
C06028=1027.667,346.518,363.481,171.794,47.266,159.278
C06029=1027.674,346.765,363.444,171.801,47.266,159.279
C06030=1027.682,347.012,363.407,171.807,47.267,159.279
C06031=1027.689,347.259,363.369,171.813,47.267,159.280
C06032=1027.697,347.506,363.332,171.820,47.268,159.281
C06033=1027.704,347.753,363.295,171.826,47.268,159.282
C06034=1027.712,348.000,363.258,171.833,47.268,159.283
C06035=1027.720,348.247,363.220,171.839,47.269,159.284
C06036=1027.728,348.494,363.183,171.845,47.270,159.285
C06037=1027.735,348.741,363.146,171.852,47.270,159.286
C06038=1027.743,348.989,363.108,171.859,47.271,159.287
C06039=1027.751,349.235,363.071,171.866,47.271,159.288
C06040=1027.759,349.483,363.033,171.872,47.272,159.289
C06041=1027.766,349.730,362.995,171.878,47.273,159.290
C06042=1027.774,349.977,362.958,171.885,47.273,159.291
C06043=1027.781,350.193,362.925,171.891,47.274,159.292
C06044=1027.787,350.409,362.892,171.896,47.275,159.293
C06045=1027.795,350.626,362.859,171.902,47.275,159.294
C06046=1027.801,350.842,362.826,171.908,47.275,159.295
C06047=1027.808,351.058,362.793,171.914,47.276,159.296
C06048=1027.815,351.275,362.759,171.920,47.276,159.296
C06049=1027.821,351.491,362.726,171.925,47.277,159.297
C06050=1027.828,351.707,362.693,171.931,47.277,159.298
C06051=1027.836,351.954,362.655,171.938,47.278,159.299
C06052=1027.844,352.201,362.618,171.944,47.279,159.300
C06053=1027.851,352.448,362.580,171.951,47.279,159.301
C06054=1027.859,352.695,362.542,171.958,47.280,159.302
C06055=1027.867,352.942,362.504,171.965,47.281,159.303
C06056=1027.876,353.190,362.466,171.971,47.282,159.304
C06057=1027.883,353.436,362.428,171.978,47.282,159.305
C06058=1027.890,353.683,362.390,171.985,47.283,159.307
C06059=1027.898,353.930,362.352,171.992,47.284,159.308
C06060=1027.907,354.177,362.314,171.999,47.284,159.309
C06061=1027.915,354.424,362.276,172.005,47.285,159.310
C06062=1027.922,354.671,362.238,172.012,47.286,159.311
C06063=1027.931,354.918,362.200,172.019,47.287,159.312
C06064=1027.938,355.165,362.163,172.026,47.288,159.313
C06065=1027.946,355.412,362.124,172.032,47.289,159.314
C06066=1027.954,355.659,362.086,172.040,47.290,159.315
C06067=1027.962,355.906,362.047,172.047,47.290,159.316
C06068=1027.970,356.152,362.009,172.053,47.291,159.317
C06069=1027.978,356.400,361.970,172.060,47.292,159.319
C06070=1027.986,356.647,361.932,172.067,47.293,159.320
C06071=1027.994,356.893,361.893,172.074,47.294,159.321
C06072=1028.002,357.141,361.855,172.081,47.295,159.322
C06073=1028.009,357.387,361.816,172.088,47.296,159.323
C06074=1028.017,357.634,361.778,172.095,47.296,159.324
C06075=1028.026,357.882,361.739,172.102,47.297,159.325
C06076=1028.033,358.128,361.701,172.108,47.298,159.326
C06077=1028.042,358.375,361.663,172.116,47.299,159.328
C06078=1028.050,358.622,361.624,172.123,47.300,159.329
C06079=1028.058,358.868,361.585,172.130,47.301,159.330
C06080=1028.066,359.115,361.547,172.137,47.302,159.331
C06081=1028.074,359.362,361.508,172.144,47.303,159.332
C06082=1028.082,359.609,361.470,172.151,47.304,159.333
C06083=1028.090,359.856,361.431,172.158,47.305,159.334
C06084=1028.098,360.103,361.392,172.165,47.306,159.336
C06085=1028.107,360.350,361.353,172.172,47.307,159.337
C06086=1028.115,360.597,361.314,172.179,47.308,159.338
C06087=1028.122,360.843,361.275,172.187,47.309,159.339
C06088=1028.130,361.090,361.236,172.194,47.310,159.340
C06089=1028.139,361.337,361.197,172.201,47.312,159.342
C06090=1028.147,361.584,361.158,172.208,47.312,159.343
C06091=1028.154,361.831,361.119,172.216,47.314,159.344
C06092=1028.162,362.077,361.080,172.222,47.315,159.345
C06093=1028.170,362.324,361.041,172.230,47.316,159.346
C06094=1028.179,362.571,361.002,172.237,47.317,159.348
C06095=1028.187,362.818,360.962,172.244,47.318,159.349
C06096=1028.195,363.065,360.923,172.252,47.319,159.350
C06097=1028.203,363.311,360.884,172.258,47.320,159.351
C06098=1028.210,363.558,360.845,172.266,47.322,159.353
C06099=1028.219,363.805,360.805,172.274,47.323,159.354
C06100=1028.227,364.052,360.767,172.281,47.324,159.355
C06101=1028.235,364.298,360.727,172.288,47.325,159.356
C06102=1028.243,364.545,360.687,172.295,47.327,159.358
C06103=1028.251,364.765,360.652,172.302,47.327,159.359
C06104=1028.258,364.984,360.618,172.309,47.329,159.360
C06105=1028.266,365.204,360.582,172.315,47.330,159.361
C06106=1028.272,365.424,360.547,172.322,47.331,159.362
C06107=1028.280,365.643,360.512,172.328,47.332,159.363
C06108=1028.288,365.862,360.477,172.335,47.333,159.365
C06109=1028.295,366.082,360.442,172.342,47.334,159.366
C06110=1028.302,366.302,360.406,172.348,47.336,159.367
C06111=1028.311,366.549,360.367,172.356,47.337,159.368
C06112=1028.319,366.795,360.328,172.363,47.338,159.369
C06113=1028.327,367.042,360.288,172.371,47.339,159.371
C06114=1028.336,367.289,360.248,172.379,47.341,159.372
C06115=1028.344,367.535,360.209,172.386,47.343,159.373
C06116=1028.352,367.782,360.168,172.394,47.344,159.375
C06117=1028.360,368.028,360.129,172.402,47.345,159.376
C06118=1028.370,368.276,360.089,172.409,47.346,159.377
C06119=1028.378,368.522,360.050,172.416,47.348,159.379
C06120=1028.386,368.768,360.009,172.424,47.349,159.380
C06121=1028.394,369.015,359.970,172.431,47.351,159.381
C06122=1028.402,369.262,359.930,172.439,47.353,159.383
C06123=1028.412,369.509,359.890,172.447,47.354,159.384
C06124=1028.419,369.755,359.850,172.454,47.355,159.385
C06125=1028.427,370.002,359.809,172.462,47.357,159.387
C06126=1028.436,370.248,359.770,172.470,47.358,159.388
C06127=1028.444,370.495,359.729,172.477,47.360,159.390
C06128=1028.453,370.741,359.689,172.485,47.362,159.391
C06129=1028.461,370.988,359.649,172.493,47.363,159.392
C06130=1028.469,371.235,359.608,172.501,47.365,159.394
C06131=1028.478,371.481,359.568,172.509,47.366,159.395
C06132=1028.486,371.728,359.528,172.516,47.368,159.397
C06133=1028.495,371.974,359.488,172.524,47.369,159.398
C06134=1028.503,372.221,359.447,172.533,47.371,159.400
C06135=1028.511,372.467,359.406,172.541,47.372,159.401
C06136=1028.521,372.714,359.366,172.549,47.374,159.403
C06137=1028.528,372.961,359.326,172.557,47.376,159.404
C06138=1028.537,373.207,359.285,172.564,47.377,159.405
C06139=1028.546,373.454,359.245,172.572,47.379,159.407
C06140=1028.554,373.700,359.204,172.580,47.381,159.408
C06141=1028.563,373.947,359.164,172.588,47.382,159.410
C06142=1028.571,374.193,359.123,172.596,47.384,159.411
C06143=1028.580,374.440,359.082,172.604,47.386,159.413
C06144=1028.589,374.686,359.042,172.612,47.388,159.414
C06145=1028.597,374.933,359.001,172.620,47.389,159.416
C06146=1028.605,375.179,358.961,172.628,47.391,159.417
C06147=1028.615,375.425,358.919,172.636,47.393,159.419
C06148=1028.623,375.672,358.879,172.645,47.394,159.420
C06149=1028.632,375.919,358.838,172.653,47.396,159.422
C06150=1028.641,376.165,358.797,172.661,47.398,159.423
C06151=1028.649,376.412,358.757,172.669,47.400,159.425
C06152=1028.659,376.658,358.716,172.677,47.402,159.426
C06153=1028.667,376.905,358.675,172.686,47.403,159.428
C06154=1028.675,377.151,358.634,172.693,47.405,159.429
C06155=1028.684,377.397,358.592,172.701,47.407,159.431
C06156=1028.693,377.644,358.551,172.709,47.409,159.433
C06157=1028.702,377.890,358.511,172.719,47.411,159.434
C06158=1028.711,378.137,358.470,172.727,47.413,159.436
C06159=1028.720,378.383,358.428,172.735,47.415,159.437
C06160=1028.728,378.629,358.387,172.743,47.416,159.439
C06161=1028.737,378.876,358.346,172.752,47.419,159.441
C06162=1028.745,379.122,358.304,172.760,47.421,159.442
C06163=1028.754,379.352,358.265,172.768,47.422,159.444
C06164=1028.761,379.582,358.227,172.776,47.424,159.445
C06165=1028.769,379.812,358.188,172.783,47.426,159.447
C06166=1028.777,380.042,358.149,172.791,47.428,159.448
C06167=1028.786,380.273,358.110,172.799,47.430,159.450
C06168=1028.794,380.503,358.071,172.807,47.432,159.451
C06169=1028.802,380.733,358.032,172.815,47.434,159.453
C06170=1028.810,380.963,357.993,172.823,47.435,159.454
C06171=1028.819,381.209,357.952,172.831,47.438,159.456
C06172=1028.828,381.456,357.910,172.839,47.440,159.458
C06173=1028.837,381.702,357.868,172.849,47.442,159.459
C06174=1028.846,381.948,357.826,172.857,47.444,159.461
C06175=1028.856,382.194,357.785,172.866,47.446,159.463
C06176=1028.865,382.441,357.744,172.874,47.448,159.464
C06177=1028.874,382.687,357.702,172.883,47.450,159.466
C06178=1028.883,382.934,357.660,172.892,47.453,159.468
C06179=1028.892,383.180,357.618,172.901,47.454,159.469
C06180=1028.900,383.426,357.577,172.909,47.457,159.471
C06181=1028.909,383.673,357.535,172.918,47.459,159.473
C06182=1028.919,383.918,357.493,172.926,47.461,159.475
C06183=1028.928,384.165,357.451,172.936,47.464,159.476
C06184=1028.936,384.411,357.409,172.944,47.466,159.478
C06185=1028.946,384.657,357.367,172.953,47.468,159.480
C06186=1028.955,384.903,357.325,172.962,47.470,159.482
C06187=1028.964,385.150,357.283,172.971,47.473,159.483
C06188=1028.973,385.396,357.240,172.980,47.475,159.485
C06189=1028.982,385.642,357.199,172.988,47.477,159.487
C06190=1028.992,385.888,357.156,172.998,47.479,159.489
C06191=1029.001,386.134,357.115,173.006,47.482,159.490
C06192=1029.010,386.380,357.072,173.015,47.484,159.492
C06193=1029.019,386.627,357.030,173.024,47.486,159.494
C06194=1029.028,386.873,356.987,173.033,47.488,159.496
C06195=1029.037,387.119,356.945,173.042,47.491,159.498
C06196=1029.046,387.365,356.902,173.052,47.493,159.499
C06197=1029.056,387.612,356.860,173.060,47.496,159.501
C06198=1029.064,387.858,356.817,173.069,47.498,159.503
C06199=1029.074,388.104,356.775,173.079,47.500,159.505
C06200=1029.083,388.350,356.732,173.087,47.503,159.507
C06201=1029.092,388.596,356.689,173.097,47.505,159.509
C06202=1029.101,388.842,356.646,173.106,47.508,159.511
C06203=1029.111,389.088,356.604,173.115,47.510,159.512
C06204=1029.120,389.334,356.561,173.124,47.513,159.514
C06205=1029.129,389.581,356.518,173.133,47.515,159.516
C06206=1029.139,389.827,356.475,173.143,47.518,159.518
C06207=1029.148,390.073,356.433,173.153,47.521,159.520
C06208=1029.157,390.318,356.389,173.161,47.523,159.522
C06209=1029.167,390.565,356.346,173.170,47.526,159.524
C06210=1029.176,390.811,356.303,173.180,47.528,159.526
C06211=1029.185,391.057,356.261,173.190,47.531,159.528
C06212=1029.195,391.303,356.217,173.199,47.534,159.530
C06213=1029.204,391.549,356.174,173.209,47.536,159.532
C06214=1029.214,391.794,356.130,173.217,47.539,159.533
C06215=1029.223,392.041,356.087,173.227,47.541,159.535
C06216=1029.232,392.287,356.045,173.236,47.544,159.537
C06217=1029.241,392.533,356.001,173.246,47.547,159.539
C06218=1029.251,392.780,355.958,173.256,47.549,159.541
C06219=1029.261,393.025,355.915,173.265,47.552,159.543
C06220=1029.270,393.271,355.870,173.275,47.555,159.545
C06221=1029.280,393.517,355.828,173.285,47.558,159.547
C06222=1029.289,393.763,355.784,173.294,47.561,159.549
C06223=1029.299,394.012,355.740,173.304,47.563,159.551
C06224=1029.308,394.262,355.695,173.314,47.567,159.554
C06225=1029.318,394.513,355.652,173.324,47.569,159.556
C06226=1029.327,394.763,355.607,173.334,47.572,159.558
C06227=1029.337,395.009,355.563,173.343,47.575,159.560
C06228=1029.347,395.255,355.519,173.353,47.578,159.562
C06229=1029.357,395.501,355.475,173.363,47.581,159.564
C06230=1029.366,395.747,355.431,173.372,47.584,159.566
C06231=1029.375,395.992,355.388,173.382,47.587,159.568
C06232=1029.385,396.238,355.344,173.392,47.589,159.570
C06233=1029.395,396.484,355.300,173.403,47.592,159.572
C06234=1029.405,396.730,355.256,173.412,47.595,159.574
C06235=1029.414,396.976,355.212,173.422,47.598,159.576
C06236=1029.424,397.222,355.168,173.432,47.601,159.579
C06237=1029.434,397.468,355.124,173.442,47.604,159.581
C06238=1029.443,397.714,355.080,173.452,47.607,159.583
C06239=1029.453,397.959,355.035,173.462,47.611,159.585
C06240=1029.463,398.205,354.992,173.473,47.613,159.587
C06241=1029.473,398.451,354.947,173.483,47.617,159.589
C06242=1029.482,398.697,354.903,173.492,47.619,159.591
C06243=1029.493,398.943,354.859,173.502,47.622,159.594
C06244=1029.502,399.188,354.814,173.513,47.625,159.596
C06245=1029.512,399.434,354.769,173.523,47.629,159.598
C06246=1029.522,399.679,354.726,173.533,47.632,159.600
C06247=1029.532,399.926,354.681,173.543,47.635,159.602
C06248=1029.542,400.172,354.637,173.554,47.638,159.605
C06249=1029.552,400.417,354.592,173.564,47.642,159.607
C06250=1029.561,400.663,354.547,173.574,47.645,159.609
C06251=1029.571,400.908,354.502,173.585,47.648,159.611
C06252=1029.581,401.153,354.458,173.595,47.651,159.614
C06253=1029.592,401.400,354.413,173.606,47.655,159.616
C06254=1029.602,401.645,354.368,173.616,47.657,159.618
C06255=1029.611,401.891,354.323,173.627,47.661,159.621
C06256=1029.622,402.137,354.278,173.638,47.664,159.623
C06257=1029.631,402.382,354.233,173.648,47.667,159.625
C06258=1029.641,402.628,354.188,173.658,47.671,159.628
C06259=1029.651,402.874,354.143,173.669,47.674,159.630
C06260=1029.661,403.120,354.098,173.679,47.678,159.632
C06261=1029.671,403.365,354.053,173.691,47.681,159.635
C06262=1029.681,403.611,354.008,173.701,47.684,159.637
C06263=1029.691,403.856,353.963,173.712,47.688,159.639
C06264=1029.701,404.102,353.918,173.722,47.691,159.642
C06265=1029.711,404.347,353.872,173.733,47.695,159.644
C06266=1029.722,404.594,353.827,173.744,47.698,159.647
C06267=1029.732,404.838,353.781,173.755,47.701,159.649
C06268=1029.742,405.085,353.736,173.766,47.705,159.651
C06269=1029.751,405.330,353.690,173.776,47.708,159.654
C06270=1029.762,405.576,353.645,173.788,47.712,159.656
C06271=1029.772,405.822,353.599,173.798,47.716,159.659
C06272=1029.782,406.067,353.553,173.809,47.719,159.661
C06273=1029.793,406.313,353.508,173.820,47.722,159.663
C06274=1029.803,406.558,353.462,173.831,47.727,159.666
C06275=1029.813,406.803,353.417,173.842,47.730,159.669
C06276=1029.824,407.050,353.371,173.854,47.733,159.671
C06277=1029.834,407.295,353.326,173.865,47.737,159.673
C06278=1029.845,407.541,353.280,173.875,47.740,159.676
C06279=1029.855,407.786,353.234,173.887,47.744,159.679
C06280=1029.865,408.031,353.188,173.898,47.748,159.681
C06281=1029.876,408.277,353.142,173.910,47.752,159.684
C06282=1029.887,408.522,353.096,173.921,47.755,159.686
C06283=1029.898,408.794,353.045,173.933,47.760,159.689
C06284=1029.910,409.066,352.995,173.946,47.763,159.692
C06285=1029.922,409.337,352.944,173.959,47.768,159.695
C06286=1029.933,409.609,352.893,173.971,47.772,159.697
C06287=1029.944,409.854,352.846,173.982,47.775,159.700
C06288=1029.955,410.100,352.800,173.994,47.779,159.703
C06289=1029.965,410.345,352.754,174.005,47.783,159.705
C06290=1029.975,410.591,352.707,174.017,47.787,159.708
C06291=1029.986,410.836,352.661,174.029,47.791,159.711
C06292=1029.997,411.081,352.615,174.040,47.795,159.713
C06293=1030.007,411.327,352.568,174.052,47.799,159.716
C06294=1030.018,411.572,352.521,174.064,47.803,159.719
C06295=1030.028,411.819,352.475,174.075,47.807,159.721
C06296=1030.039,412.064,352.428,174.087,47.811,159.724
C06297=1030.050,412.309,352.381,174.099,47.815,159.727
C06298=1030.060,412.554,352.334,174.110,47.819,159.729
C06299=1030.071,412.799,352.287,174.122,47.822,159.732
C06300=1030.082,413.045,352.241,174.135,47.827,159.735
C06301=1030.093,413.290,352.194,174.147,47.831,159.738
C06302=1030.104,413.535,352.147,174.158,47.834,159.740
C06303=1030.114,413.781,352.100,174.170,47.839,159.743
C06304=1030.125,414.026,352.053,174.182,47.843,159.746
C06305=1030.136,414.272,352.006,174.195,47.847,159.749
C06306=1030.147,414.517,351.959,174.207,47.851,159.751
C06307=1030.158,414.762,351.912,174.219,47.855,159.754
C06308=1030.169,415.008,351.864,174.231,47.860,159.757
C06309=1030.180,415.253,351.817,174.243,47.863,159.760
C06310=1030.191,415.499,351.770,174.255,47.868,159.763
C06311=1030.202,415.743,351.723,174.267,47.872,159.766
C06312=1030.214,415.989,351.676,174.280,47.876,159.769
C06313=1030.224,416.234,351.628,174.292,47.881,159.772
C06314=1030.236,416.479,351.581,174.305,47.884,159.774
C06315=1030.246,416.724,351.533,174.317,47.889,159.777
C06316=1030.258,416.969,351.486,174.329,47.894,159.780
C06317=1030.269,417.215,351.437,174.342,47.898,159.783
C06318=1030.279,417.460,351.390,174.354,47.902,159.786
C06319=1030.291,417.705,351.342,174.367,47.906,159.789
C06320=1030.302,417.950,351.294,174.379,47.911,159.792
C06321=1030.312,418.195,351.246,174.393,47.915,159.795
C06322=1030.324,418.440,351.199,174.405,47.920,159.798
C06323=1030.335,418.685,351.150,174.418,47.924,159.801
C06324=1030.346,418.931,351.102,174.431,47.928,159.804
C06325=1030.358,419.176,351.054,174.443,47.933,159.807
C06326=1030.369,419.421,351.006,174.457,47.937,159.810
C06327=1030.380,419.666,350.958,174.470,47.942,159.813
C06328=1030.391,419.911,350.910,174.482,47.946,159.816
C06329=1030.403,420.156,350.862,174.495,47.951,159.819
C06330=1030.414,420.401,350.813,174.509,47.956,159.823
C06331=1030.425,420.646,350.765,174.521,47.960,159.825
C06332=1030.437,420.891,350.717,174.534,47.965,159.829
C06333=1030.448,421.137,350.669,174.547,47.969,159.832
C06334=1030.460,421.382,350.620,174.561,47.974,159.835
C06335=1030.471,421.627,350.572,174.574,47.978,159.838
C06336=1030.483,421.871,350.523,174.588,47.983,159.841
C06337=1030.494,422.117,350.475,174.601,47.988,159.844
C06338=1030.507,422.362,350.426,174.613,47.992,159.847
C06339=1030.518,422.607,350.377,174.627,47.997,159.851
C06340=1030.529,422.852,350.329,174.640,48.002,159.854
C06341=1030.541,423.097,350.280,174.654,48.007,159.857
C06342=1030.552,423.341,350.231,174.667,48.011,159.860
C06343=1030.570,423.704,350.158,174.688,48.018,159.865
C06344=1030.587,424.065,350.086,174.708,48.026,159.870
C06345=1030.604,424.428,350.013,174.729,48.033,159.875
C06346=1030.622,424.788,349.940,174.749,48.040,159.880
C06347=1030.634,425.034,349.891,174.762,48.045,159.883
C06348=1030.645,425.279,349.842,174.776,48.050,159.887
C06349=1030.657,425.524,349.793,174.790,48.055,159.890
C06350=1030.669,425.768,349.743,174.804,48.060,159.893
C06351=1030.689,426.178,349.660,174.827,48.069,159.899
C06352=1030.708,426.588,349.578,174.851,48.077,159.905
C06353=1030.729,426.998,349.494,174.875,48.085,159.911
C06354=1030.749,427.407,349.411,174.898,48.094,159.916
C06355=1030.761,427.652,349.361,174.913,48.099,159.920
C06356=1030.773,427.896,349.311,174.927,48.104,159.923
C06357=1030.785,428.141,349.261,174.942,48.109,159.927
C06358=1030.797,428.385,349.211,174.956,48.114,159.931
C06359=1030.809,428.631,349.160,174.971,48.119,159.934
C06360=1030.821,428.875,349.110,174.985,48.125,159.938
C06361=1030.833,429.120,349.060,175.000,48.130,159.941
C06362=1030.845,429.364,349.010,175.015,48.135,159.945
C06363=1030.858,429.609,348.960,175.029,48.141,159.948
C06364=1030.870,429.854,348.910,175.044,48.146,159.952
C06365=1030.882,430.098,348.859,175.059,48.151,159.956
C06366=1030.894,430.343,348.808,175.074,48.157,159.959
C06367=1030.907,430.588,348.758,175.089,48.162,159.963
C06368=1030.919,430.832,348.707,175.104,48.167,159.967
C06369=1030.932,431.077,348.657,175.119,48.173,159.970
C06370=1030.944,431.321,348.607,175.133,48.178,159.974
C06371=1030.957,431.566,348.556,175.148,48.184,159.978
C06372=1030.969,431.810,348.506,175.164,48.189,159.982
C06373=1030.981,432.055,348.454,175.179,48.194,159.985
C06374=1030.993,432.299,348.403,175.194,48.200,159.989
C06375=1031.006,432.543,348.353,175.209,48.205,159.993
C06376=1031.019,432.788,348.301,175.225,48.211,159.997
C06377=1031.032,433.032,348.251,175.240,48.217,160.001
C06378=1031.044,433.277,348.200,175.256,48.222,160.004
C06379=1031.058,433.522,348.149,175.271,48.227,160.008
C06380=1031.070,433.766,348.097,175.287,48.233,160.012
C06381=1031.083,434.011,348.046,175.303,48.239,160.016
C06382=1031.095,434.255,347.995,175.318,48.244,160.020
C06383=1031.108,434.499,347.943,175.334,48.250,160.024
C06384=1031.121,434.744,347.892,175.350,48.256,160.028
C06385=1031.133,434.988,347.841,175.366,48.262,160.032
C06386=1031.146,435.233,347.789,175.382,48.267,160.036
C06387=1031.159,435.477,347.738,175.397,48.273,160.040
C06388=1031.172,435.721,347.686,175.414,48.279,160.044
C06389=1031.185,435.966,347.633,175.430,48.285,160.048
C06390=1031.198,436.210,347.583,175.445,48.291,160.052
C06391=1031.211,436.455,347.530,175.462,48.296,160.056
C06392=1031.224,436.699,347.478,175.478,48.303,160.060
C06393=1031.237,436.942,347.427,175.494,48.308,160.064
C06394=1031.250,437.187,347.374,175.510,48.314,160.068
C06395=1031.263,437.431,347.322,175.527,48.320,160.072
C06396=1031.275,437.675,347.270,175.544,48.326,160.076
C06397=1031.289,437.920,347.218,175.560,48.332,160.080
C06398=1031.302,438.163,347.165,175.577,48.338,160.085
C06399=1031.317,438.427,347.109,175.595,48.344,160.089
C06400=1031.331,438.690,347.053,175.613,48.351,160.094
C06401=1031.345,438.953,346.996,175.631,48.357,160.098
C06402=1031.359,439.216,346.940,175.649,48.364,160.103
C06403=1031.372,439.460,346.887,175.666,48.370,160.107
C06404=1031.386,439.704,346.834,175.683,48.376,160.111
C06405=1031.400,439.949,346.781,175.700,48.383,160.116
C06406=1031.413,440.193,346.729,175.717,48.389,160.120
C06407=1031.426,440.437,346.676,175.734,48.395,160.125
C06408=1031.440,440.680,346.623,175.751,48.401,160.129
C06409=1031.453,440.924,346.570,175.768,48.407,160.133
C06410=1031.467,441.168,346.517,175.786,48.413,160.138
C06411=1031.480,441.412,346.464,175.803,48.420,160.142
C06412=1031.494,441.657,346.410,175.822,48.426,160.147
C06413=1031.508,441.900,346.358,175.839,48.432,160.151
C06414=1031.521,442.144,346.305,175.856,48.439,160.155
C06415=1031.536,442.388,346.251,175.874,48.445,160.160
C06416=1031.549,442.632,346.198,175.892,48.451,160.165
C06417=1031.563,442.876,346.145,175.909,48.458,160.169
C06418=1031.577,443.120,346.091,175.927,48.464,160.174
C06419=1031.591,443.363,346.038,175.945,48.471,160.178
C06420=1031.605,443.606,345.984,175.963,48.478,160.183
C06421=1031.620,443.849,345.932,175.981,48.483,160.187
C06422=1031.635,444.093,345.880,176.000,48.490,160.192
C06423=1031.650,444.336,345.828,176.018,48.496,160.196
C06424=1031.667,444.579,345.776,176.035,48.502,160.201
C06425=1031.683,444.823,345.726,176.054,48.508,160.206
C06426=1031.701,445.067,345.675,176.073,48.514,160.210
C06427=1031.718,445.311,345.625,176.091,48.519,160.214
C06428=1031.737,445.555,345.576,176.109,48.525,160.219
C06429=1031.756,445.798,345.526,176.129,48.530,160.223
C06430=1031.775,446.042,345.477,176.147,48.537,160.228
C06431=1031.795,446.287,345.429,176.167,48.542,160.233
C06432=1031.815,446.531,345.381,176.185,48.547,160.237
C06433=1031.835,446.775,345.333,176.205,48.552,160.241
C06434=1031.857,447.020,345.286,176.224,48.558,160.246
C06435=1031.879,447.264,345.239,176.243,48.563,160.250
C06436=1031.901,447.509,345.192,176.262,48.569,160.255
C06437=1031.924,447.753,345.147,176.281,48.573,160.259
C06438=1031.947,447.998,345.101,176.301,48.578,160.264
C06439=1031.971,448.243,345.056,176.320,48.584,160.268
C06440=1031.995,448.487,345.011,176.340,48.588,160.272
C06441=1032.019,448.733,344.967,176.360,48.593,160.277
C06442=1032.045,448.977,344.923,176.379,48.598,160.281
C06443=1032.070,449.223,344.879,176.399,48.602,160.286
C06444=1032.097,449.468,344.836,176.419,48.607,160.290
C06445=1032.124,449.713,344.794,176.440,48.611,160.294
C06446=1032.150,449.958,344.751,176.460,48.615,160.299
C06447=1032.178,450.204,344.709,176.480,48.620,160.303
C06448=1032.206,450.449,344.669,176.501,48.624,160.308
C06449=1032.235,450.694,344.627,176.520,48.629,160.312
C06450=1032.265,450.939,344.587,176.541,48.633,160.316
C06451=1032.293,451.185,344.547,176.562,48.637,160.321
C06452=1032.324,451.431,344.507,176.583,48.640,160.325
C06453=1032.355,451.675,344.467,176.603,48.644,160.329
C06454=1032.386,451.921,344.429,176.624,48.648,160.334
C06455=1032.418,452.167,344.391,176.645,48.652,160.338
C06456=1032.450,452.413,344.352,176.666,48.656,160.342
C06457=1032.483,452.658,344.315,176.687,48.660,160.347
C06458=1032.516,452.903,344.278,176.708,48.664,160.351
C06459=1032.573,453.314,344.217,176.745,48.669,160.358
C06460=1032.290,453.381,343.886,176.748,48.734,160.379
C06461=1032.239,453.015,343.940,176.715,48.730,160.373
C06462=1032.206,452.770,343.977,176.695,48.726,160.368
C06463=1032.173,452.524,344.014,176.673,48.722,160.364
C06464=1032.141,452.279,344.052,176.652,48.718,160.360
C06465=1032.109,452.033,344.090,176.631,48.715,160.355
C06466=1032.077,451.787,344.128,176.610,48.711,160.351
C06467=1032.046,451.542,344.168,176.589,48.708,160.347
C06468=1032.016,451.297,344.207,176.568,48.704,160.342
C06469=1031.986,451.051,344.248,176.548,48.700,160.338
C06470=1031.956,450.806,344.288,176.527,48.696,160.334
C06471=1031.927,450.560,344.328,176.506,48.692,160.329
C06472=1031.899,450.315,344.369,176.486,48.687,160.325
C06473=1031.871,450.070,344.411,176.465,48.683,160.321
C06474=1031.844,449.824,344.453,176.445,48.679,160.316
C06475=1031.817,449.579,344.496,176.425,48.674,160.312
C06476=1031.790,449.334,344.538,176.406,48.670,160.307
C06477=1031.764,449.088,344.581,176.385,48.666,160.303
C06478=1031.738,448.845,344.625,176.366,48.661,160.299
C06479=1031.713,448.599,344.669,176.346,48.656,160.294
C06480=1031.689,448.354,344.714,176.326,48.652,160.290
C06481=1031.665,448.110,344.759,176.306,48.647,160.285
C06482=1031.641,447.865,344.804,176.287,48.642,160.281
C06483=1031.619,447.620,344.850,176.267,48.637,160.277
C06484=1031.597,447.375,344.896,176.247,48.632,160.272
C06485=1031.574,447.131,344.942,176.229,48.627,160.268
C06486=1031.553,446.886,344.990,176.209,48.622,160.263
C06487=1031.531,446.642,345.037,176.190,48.616,160.259
C06488=1031.511,446.398,345.084,176.171,48.612,160.254
C06489=1031.491,446.153,345.133,176.152,48.606,160.250
C06490=1031.471,445.909,345.181,176.133,48.601,160.245
C06491=1031.452,445.665,345.230,176.114,48.595,160.241
C06492=1031.434,445.421,345.280,176.095,48.590,160.236
C06493=1031.416,445.178,345.329,176.077,48.584,160.232
C06494=1031.398,444.934,345.380,176.059,48.578,160.228
C06495=1031.381,444.689,345.431,176.039,48.572,160.223
C06496=1031.364,444.446,345.482,176.021,48.566,160.218
C06497=1031.348,444.203,345.533,176.003,48.560,160.214
C06498=1031.333,443.959,345.585,175.985,48.554,160.209
C06499=1031.318,443.715,345.638,175.967,48.548,160.205
C06500=1031.303,443.472,345.690,175.948,48.542,160.200
C06501=1031.289,443.230,345.743,175.931,48.535,160.196
C06502=1031.275,442.986,345.797,175.913,48.530,160.191
C06503=1031.262,442.742,345.850,175.895,48.523,160.186
C06504=1031.247,442.499,345.904,175.877,48.517,160.182
C06505=1031.234,442.255,345.957,175.859,48.511,160.178
C06506=1031.219,442.010,346.010,175.842,48.504,160.173
C06507=1031.206,441.766,346.063,175.823,48.498,160.169
C06508=1031.193,441.523,346.117,175.806,48.492,160.164
C06509=1031.179,441.279,346.170,175.789,48.486,160.160
C06510=1031.165,441.035,346.223,175.772,48.479,160.155
C06511=1031.151,440.791,346.276,175.754,48.473,160.151
C06512=1031.138,440.547,346.329,175.737,48.467,160.146
C06513=1031.125,440.303,346.381,175.719,48.461,160.142
C06514=1031.112,440.059,346.434,175.702,48.455,160.138
C06515=1031.098,439.815,346.487,175.685,48.449,160.133
C06516=1031.085,439.571,346.540,175.668,48.443,160.129
C06517=1031.071,439.327,346.592,175.652,48.436,160.125
C06518=1031.057,439.063,346.650,175.633,48.430,160.120
C06519=1031.042,438.799,346.706,175.615,48.424,160.116
C06520=1031.029,438.535,346.762,175.596,48.417,160.111
C06521=1031.013,438.271,346.820,175.579,48.411,160.107
C06522=1031.000,438.026,346.872,175.562,48.405,160.102
C06523=1030.988,437.783,346.924,175.545,48.399,160.098
C06524=1030.975,437.538,346.976,175.528,48.394,160.094
C06525=1030.961,437.294,347.028,175.512,48.387,160.090
C06526=1030.948,437.049,347.080,175.496,48.382,160.086
C06527=1030.935,436.806,347.132,175.480,48.375,160.082
C06528=1030.922,436.561,347.184,175.463,48.370,160.078
C06529=1030.909,436.317,347.236,175.447,48.364,160.074
C06530=1030.896,436.073,347.288,175.430,48.358,160.069
C06531=1030.883,435.829,347.340,175.415,48.352,160.065
C06532=1030.870,435.584,347.392,175.398,48.347,160.062
C06533=1030.857,435.340,347.443,175.382,48.341,160.057
C06534=1030.844,435.095,347.494,175.366,48.336,160.053
C06535=1030.832,434.851,347.546,175.350,48.330,160.050
C06536=1030.819,434.606,347.598,175.335,48.324,160.046
C06537=1030.806,434.363,347.649,175.318,48.319,160.042
C06538=1030.793,434.118,347.701,175.303,48.313,160.038
C06539=1030.781,433.873,347.752,175.287,48.308,160.034
C06540=1030.768,433.630,347.803,175.272,48.302,160.030
C06541=1030.755,433.385,347.855,175.256,48.296,160.026
C06542=1030.743,433.140,347.906,175.240,48.291,160.022
C06543=1030.730,432.896,347.957,175.225,48.286,160.018
C06544=1030.717,432.651,348.008,175.209,48.280,160.015
C06545=1030.704,432.406,348.058,175.194,48.275,160.011
C06546=1030.692,432.162,348.109,175.179,48.269,160.007
C06547=1030.679,431.918,348.159,175.163,48.264,160.003
C06548=1030.666,431.673,348.211,175.148,48.259,160.000
C06549=1030.654,431.428,348.261,175.133,48.253,159.996
C06550=1030.642,431.184,348.312,175.118,48.248,159.992
C06551=1030.629,430.940,348.363,175.103,48.243,159.988
C06552=1030.617,430.695,348.413,175.088,48.237,159.985
C06553=1030.605,430.450,348.463,175.073,48.232,159.981
C06554=1030.592,430.206,348.514,175.058,48.227,159.977
C06555=1030.580,429.961,348.564,175.043,48.221,159.974
C06556=1030.567,429.717,348.615,175.028,48.216,159.970
C06557=1030.555,429.472,348.666,175.014,48.211,159.966
C06558=1030.544,429.227,348.715,174.999,48.206,159.963
C06559=1030.531,428.983,348.765,174.984,48.201,159.959
C06560=1030.519,428.738,348.815,174.970,48.195,159.956
C06561=1030.507,428.493,348.866,174.955,48.190,159.952
C06562=1030.494,428.248,348.916,174.941,48.185,159.949
C06563=1030.483,428.004,348.965,174.926,48.180,159.945
C06564=1030.471,427.759,349.016,174.912,48.175,159.942
C06565=1030.459,427.514,349.066,174.897,48.170,159.938
C06566=1030.447,427.270,349.116,174.883,48.165,159.935
C06567=1030.435,427.025,349.166,174.869,48.160,159.931
C06568=1030.423,426.780,349.215,174.855,48.155,159.928
C06569=1030.411,426.536,349.265,174.840,48.150,159.924
C06570=1030.399,426.290,349.314,174.826,48.145,159.921
C06571=1030.387,426.046,349.364,174.813,48.140,159.917
C06572=1030.375,425.801,349.414,174.798,48.135,159.914
C06573=1030.364,425.556,349.463,174.784,48.130,159.911
C06574=1030.351,425.311,349.512,174.770,48.125,159.907
C06575=1030.340,425.067,349.561,174.755,48.120,159.904
C06576=1030.328,424.821,349.610,174.742,48.116,159.901
C06577=1030.316,424.577,349.660,174.728,48.111,159.897
C06578=1030.303,424.293,349.717,174.712,48.105,159.893
C06579=1030.288,424.008,349.774,174.697,48.100,159.890
C06580=1030.275,423.724,349.831,174.680,48.094,159.886
C06581=1030.262,423.440,349.888,174.665,48.088,159.882
C06582=1030.250,423.196,349.937,174.652,48.084,159.879
C06583=1030.238,422.950,349.986,174.638,48.079,159.875
C06584=1030.227,422.705,350.035,174.624,48.075,159.872
C06585=1030.216,422.460,350.083,174.610,48.070,159.869
C06586=1030.204,422.215,350.132,174.597,48.065,159.866
C06587=1030.192,421.970,350.180,174.584,48.060,159.863
C06588=1030.180,421.725,350.229,174.571,48.056,159.859
C06589=1030.169,421.479,350.278,174.558,48.052,159.856
C06590=1030.157,421.235,350.326,174.544,48.047,159.853
C06591=1030.146,420.990,350.374,174.531,48.043,159.850
C06592=1030.135,420.745,350.423,174.518,48.038,159.847
C06593=1030.123,420.500,350.471,174.504,48.033,159.844
C06594=1030.112,420.254,350.519,174.491,48.029,159.841
C06595=1030.100,420.010,350.568,174.479,48.025,159.838
C06596=1030.088,419.765,350.616,174.466,48.020,159.835
C06597=1030.077,419.519,350.664,174.452,48.016,159.831
C06598=1030.060,419.140,350.738,174.433,48.009,159.827
C06599=1030.043,418.761,350.813,174.412,48.003,159.822
C06600=1030.025,418.381,350.887,174.393,47.995,159.817
C06601=1030.008,418.001,350.961,174.374,47.989,159.813
C06602=1029.997,417.757,351.009,174.360,47.984,159.810
C06603=1029.986,417.511,351.057,174.347,47.980,159.807
C06604=1029.975,417.266,351.105,174.335,47.976,159.804
C06605=1029.964,417.021,351.153,174.322,47.972,159.801
C06606=1029.953,416.775,351.200,174.310,47.967,159.798
C06607=1029.942,416.531,351.248,174.297,47.963,159.795
C06608=1029.931,416.285,351.295,174.285,47.959,159.792
C06609=1029.920,416.040,351.343,174.273,47.955,159.790
C06610=1029.909,415.795,351.390,174.260,47.951,159.787
C06611=1029.897,415.549,351.437,174.248,47.946,159.784
C06612=1029.887,415.304,351.485,174.235,47.942,159.781
C06613=1029.875,415.059,351.532,174.224,47.938,159.778
C06614=1029.865,414.814,351.579,174.212,47.934,159.775
C06615=1029.853,414.568,351.626,174.199,47.930,159.772
C06616=1029.842,414.323,351.673,174.187,47.926,159.769
C06617=1029.832,414.077,351.720,174.175,47.922,159.767
C06618=1029.821,413.832,351.767,174.162,47.918,159.764
C06619=1029.811,413.587,351.814,174.150,47.914,159.761
C06620=1029.799,413.341,351.861,174.139,47.910,159.758
C06621=1029.788,413.096,351.908,174.127,47.906,159.756
C06622=1029.778,412.851,351.955,174.115,47.902,159.753
C06623=1029.767,412.606,352.002,174.102,47.898,159.750
C06624=1029.755,412.360,352.049,174.091,47.894,159.747
C06625=1029.745,412.115,352.096,174.079,47.891,159.745
C06626=1029.735,411.869,352.142,174.067,47.887,159.742
C06627=1029.724,411.624,352.189,174.056,47.883,159.739
C06628=1029.714,411.379,352.236,174.044,47.879,159.737
C06629=1029.703,411.133,352.282,174.032,47.875,159.734
C06630=1029.693,410.888,352.329,174.021,47.871,159.731
C06631=1029.682,410.642,352.375,174.009,47.867,159.729
C06632=1029.671,410.396,352.422,173.998,47.864,159.726
C06633=1029.661,410.151,352.468,173.986,47.860,159.723
C06634=1029.644,409.767,352.541,173.967,47.854,159.719
C06635=1029.627,409.382,352.612,173.950,47.848,159.715
C06636=1029.610,408.997,352.685,173.931,47.843,159.711
C06637=1029.594,408.612,352.756,173.914,47.837,159.707
C06638=1029.583,408.366,352.802,173.902,47.833,159.705
C06639=1029.573,408.121,352.848,173.891,47.830,159.702
C06640=1029.563,407.875,352.895,173.880,47.826,159.700
C06641=1029.552,407.629,352.941,173.868,47.823,159.697
C06642=1029.542,407.384,352.986,173.858,47.819,159.695
C06643=1029.532,407.139,353.032,173.846,47.815,159.692
C06644=1029.521,406.893,353.078,173.835,47.812,159.690
C06645=1029.510,406.648,353.124,173.824,47.808,159.687
C06646=1029.501,406.402,353.169,173.813,47.805,159.685
C06647=1029.490,406.156,353.215,173.802,47.801,159.682
C06648=1029.479,405.911,353.260,173.791,47.798,159.680
C06649=1029.470,405.665,353.305,173.779,47.795,159.677
C06650=1029.459,405.420,353.351,173.769,47.791,159.675
C06651=1029.449,405.174,353.396,173.758,47.788,159.672
C06652=1029.439,404.929,353.442,173.747,47.784,159.670
C06653=1029.428,404.682,353.487,173.736,47.781,159.668
C06654=1029.418,404.438,353.533,173.725,47.778,159.665
C06655=1029.408,404.191,353.578,173.715,47.774,159.663
C06656=1029.398,403.946,353.623,173.704,47.770,159.660
C06657=1029.388,403.700,353.669,173.694,47.767,159.658
C06658=1029.378,403.455,353.713,173.682,47.764,159.656
C06659=1029.368,403.210,353.759,173.671,47.761,159.654
C06660=1029.358,402.964,353.804,173.661,47.757,159.651
C06661=1029.348,402.718,353.849,173.650,47.754,159.649
C06662=1029.338,402.473,353.894,173.640,47.751,159.646
C06663=1029.329,402.226,353.940,173.630,47.748,159.644
C06664=1029.319,401.981,353.984,173.618,47.744,159.642
C06665=1029.308,401.735,354.029,173.608,47.741,159.640
C06666=1029.298,401.489,354.074,173.597,47.738,159.637
C06667=1029.288,401.244,354.119,173.587,47.734,159.635
C06668=1029.279,400.998,354.163,173.576,47.732,159.633
C06669=1029.269,400.753,354.208,173.566,47.728,159.630
C06670=1029.259,400.506,354.253,173.556,47.725,159.628
C06671=1029.249,400.261,354.297,173.545,47.722,159.626
C06672=1029.239,400.015,354.342,173.535,47.719,159.624
C06673=1029.229,399.769,354.387,173.525,47.716,159.622
C06674=1029.220,399.523,354.431,173.514,47.713,159.619
C06675=1029.210,399.278,354.476,173.504,47.710,159.617
C06676=1029.199,399.033,354.520,173.494,47.707,159.615
C06677=1029.190,398.787,354.564,173.483,47.704,159.613
C06678=1029.180,398.540,354.609,173.473,47.701,159.610
C06679=1029.170,398.294,354.653,173.464,47.698,159.608
C06680=1029.160,398.048,354.697,173.454,47.695,159.606
C06681=1029.150,397.803,354.741,173.443,47.692,159.604
C06682=1029.140,397.557,354.785,173.433,47.689,159.602
C06683=1029.131,397.311,354.829,173.423,47.686,159.600
C06684=1029.120,397.066,354.873,173.413,47.683,159.598
C06685=1029.111,396.820,354.917,173.403,47.681,159.596
C06686=1029.102,396.573,354.962,173.393,47.677,159.593
C06687=1029.092,396.328,355.005,173.383,47.675,159.591
C06688=1029.083,396.082,355.049,173.373,47.672,159.589
C06689=1029.073,395.836,355.093,173.363,47.669,159.587
C06690=1029.063,395.590,355.136,173.353,47.666,159.585
C06691=1029.054,395.344,355.181,173.344,47.663,159.583
C06692=1029.044,395.098,355.224,173.334,47.660,159.581
C06693=1029.035,394.853,355.268,173.324,47.657,159.579
C06694=1029.025,394.601,355.313,173.314,47.655,159.577
C06695=1029.015,394.348,355.358,173.304,47.652,159.575
C06696=1029.005,394.096,355.402,173.294,47.649,159.573
C06697=1028.995,393.843,355.447,173.284,47.646,159.571
C06698=1028.986,393.598,355.491,173.275,47.644,159.569
C06699=1028.976,393.351,355.534,173.265,47.641,159.567
C06700=1028.967,393.105,355.578,173.256,47.638,159.565
C06701=1028.958,392.860,355.620,173.246,47.636,159.563
C06702=1028.948,392.613,355.664,173.236,47.633,159.561
C06703=1028.938,392.368,355.708,173.227,47.631,159.559
C06704=1028.929,392.122,355.750,173.217,47.628,159.557
C06705=1028.920,391.875,355.794,173.207,47.625,159.555
C06706=1028.910,391.629,355.837,173.198,47.623,159.553
C06707=1028.901,391.383,355.880,173.188,47.620,159.551
C06708=1028.891,391.137,355.924,173.179,47.617,159.549
C06709=1028.882,390.892,355.966,173.169,47.615,159.547
C06710=1028.873,390.645,356.009,173.160,47.613,159.545
C06711=1028.863,390.400,356.053,173.151,47.610,159.543
C06712=1028.854,390.153,356.096,173.142,47.607,159.541
C06713=1028.845,389.907,356.138,173.132,47.605,159.539
C06714=1028.836,389.662,356.181,173.122,47.602,159.537
C06715=1028.827,389.415,356.224,173.113,47.600,159.535
C06716=1028.817,389.169,356.267,173.104,47.597,159.533
C06717=1028.807,388.923,356.309,173.095,47.595,159.532
C06718=1028.799,388.677,356.352,173.086,47.593,159.530
C06719=1028.790,388.431,356.395,173.076,47.590,159.528
C06720=1028.780,388.184,356.438,173.067,47.588,159.526
C06721=1028.771,387.939,356.480,173.058,47.585,159.524
C06722=1028.762,387.693,356.523,173.049,47.583,159.522
C06723=1028.752,387.446,356.566,173.040,47.581,159.521
C06724=1028.743,387.200,356.608,173.031,47.579,159.519
C06725=1028.734,386.954,356.650,173.022,47.576,159.517
C06726=1028.726,386.708,356.693,173.013,47.574,159.515
C06727=1028.716,386.461,356.735,173.003,47.572,159.513
C06728=1028.707,386.215,356.778,172.995,47.569,159.512
C06729=1028.698,385.969,356.820,172.986,47.567,159.510
C06730=1028.688,385.722,356.862,172.977,47.565,159.508
C06731=1028.679,385.476,356.904,172.968,47.563,159.506
C06732=1028.670,385.230,356.946,172.959,47.561,159.504
C06733=1028.661,384.984,356.988,172.950,47.558,159.503
C06734=1028.652,384.738,357.030,172.941,47.556,159.501
C06735=1028.643,384.492,357.072,172.932,47.554,159.499
C06736=1028.634,384.245,357.114,172.924,47.551,159.497
C06737=1028.624,383.999,357.157,172.915,47.550,159.496
C06738=1028.615,383.753,357.198,172.906,47.548,159.494
C06739=1028.606,383.506,357.240,172.897,47.545,159.492
C06740=1028.597,383.260,357.282,172.888,47.543,159.491
C06741=1028.588,383.014,357.324,172.880,47.541,159.489
C06742=1028.579,382.768,357.366,172.871,47.539,159.487
C06743=1028.570,382.521,357.408,172.862,47.537,159.486
C06744=1028.560,382.275,357.449,172.853,47.535,159.484
C06745=1028.551,382.029,357.491,172.845,47.533,159.482
C06746=1028.543,381.783,357.532,172.836,47.531,159.480
C06747=1028.534,381.536,357.574,172.828,47.529,159.479
C06748=1028.525,381.291,357.615,172.819,47.527,159.477
C06749=1028.516,381.044,357.657,172.811,47.525,159.476
C06750=1028.508,380.813,357.696,172.803,47.523,159.474
C06751=1028.500,380.581,357.736,172.795,47.521,159.473
C06752=1028.492,380.350,357.775,172.787,47.519,159.471
C06753=1028.483,380.118,357.813,172.779,47.518,159.469
C06754=1028.475,379.888,357.852,172.771,47.516,159.468
C06755=1028.467,379.657,357.891,172.763,47.514,159.466
C06756=1028.459,379.425,357.930,172.755,47.512,159.465
C06757=1028.451,379.195,357.969,172.747,47.510,159.463
C06758=1028.442,378.948,358.010,172.738,47.509,159.462
C06759=1028.433,378.702,358.052,172.730,47.507,159.460
C06760=1028.425,378.455,358.093,172.722,47.504,159.458
C06761=1028.416,378.209,358.134,172.713,47.503,159.457
C06762=1028.407,377.963,358.176,172.705,47.501,159.455
C06763=1028.399,377.716,358.217,172.697,47.499,159.454
C06764=1028.390,377.470,358.258,172.688,47.498,159.452
C06765=1028.382,377.223,358.299,172.680,47.496,159.451
C06766=1028.372,376.977,358.340,172.672,47.494,159.449
C06767=1028.364,376.731,358.381,172.664,47.492,159.448
C06768=1028.355,376.484,358.422,172.655,47.490,159.446
C06769=1028.346,376.237,358.462,172.647,47.489,159.445
C06770=1028.338,375.991,358.504,172.639,47.487,159.443
C06771=1028.328,375.745,358.544,172.630,47.485,159.441
C06772=1028.320,375.498,358.585,172.622,47.483,159.440
C06773=1028.312,375.251,358.626,172.615,47.482,159.439
C06774=1028.302,375.005,358.666,172.607,47.480,159.437
C06775=1028.294,374.758,358.707,172.598,47.479,159.436
C06776=1028.286,374.511,358.748,172.590,47.477,159.434
C06777=1028.277,374.265,358.788,172.582,47.475,159.433
C06778=1028.268,374.018,358.829,172.574,47.474,159.431
C06779=1028.259,373.772,358.869,172.566,47.472,159.430
C06780=1028.251,373.525,358.910,172.559,47.470,159.428
C06781=1028.243,373.279,358.951,172.550,47.469,159.427
C06782=1028.234,373.033,358.991,172.542,47.467,159.425
C06783=1028.225,372.786,359.032,172.534,47.466,159.424
C06784=1028.217,372.540,359.072,172.526,47.464,159.422
C06785=1028.208,372.293,359.113,172.519,47.463,159.421
C06786=1028.200,372.046,359.153,172.511,47.461,159.419
C06787=1028.192,371.800,359.193,172.503,47.459,159.418
C06788=1028.183,371.553,359.234,172.494,47.458,159.417
C06789=1028.175,371.307,359.274,172.487,47.457,159.415
C06790=1028.166,371.060,359.314,172.479,47.455,159.414
C06791=1028.158,370.813,359.355,172.471,47.453,159.412
C06792=1028.149,370.567,359.394,172.463,47.452,159.411
C06793=1028.141,370.321,359.435,172.456,47.451,159.410
C06794=1028.133,370.074,359.475,172.448,47.449,159.408
C06795=1028.124,369.827,359.515,172.440,47.448,159.407
C06796=1028.116,369.581,359.555,172.433,47.446,159.406
C06797=1028.108,369.334,359.595,172.425,47.445,159.404
C06798=1028.100,369.088,359.635,172.417,47.443,159.403
C06799=1028.092,368.841,359.675,172.409,47.442,159.401
C06800=1028.083,368.594,359.715,172.402,47.441,159.400
C06801=1028.074,368.348,359.755,172.394,47.439,159.399
C06802=1028.066,368.101,359.794,172.387,47.438,159.397
C06803=1028.058,367.854,359.834,172.379,47.437,159.396
C06804=1028.050,367.608,359.874,172.371,47.435,159.395
C06805=1028.041,367.361,359.913,172.364,47.434,159.393
C06806=1028.033,367.113,359.953,172.356,47.433,159.392
C06807=1028.024,366.867,359.993,172.348,47.431,159.391
C06808=1028.016,366.621,360.033,172.341,47.430,159.389
C06809=1028.007,366.374,360.072,172.333,47.429,159.388
C06810=1028.001,366.154,360.108,172.327,47.428,159.387
C06811=1027.993,365.933,360.143,172.320,47.427,159.386
C06812=1027.985,365.712,360.178,172.313,47.426,159.385
C06813=1027.978,365.491,360.213,172.307,47.425,159.383
C06814=1027.970,365.271,360.248,172.300,47.424,159.382
C06815=1027.964,365.050,360.284,172.293,47.423,159.381
C06816=1027.956,364.829,360.319,172.286,47.421,159.380
C06817=1027.949,364.609,360.354,172.280,47.420,159.379
C06818=1027.940,364.362,360.393,172.273,47.420,159.378
C06819=1027.932,364.116,360.433,172.265,47.418,159.376
C06820=1027.924,363.869,360.473,172.258,47.417,159.375
C06821=1027.916,363.621,360.511,172.250,47.416,159.374
C06822=1027.907,363.375,360.551,172.244,47.415,159.373
C06823=1027.900,363.128,360.590,172.236,47.413,159.371
C06824=1027.891,362.881,360.630,172.229,47.413,159.370
C06825=1027.884,362.635,360.668,172.221,47.411,159.369
C06826=1027.875,362.388,360.707,172.214,47.411,159.368
C06827=1027.867,362.141,360.747,172.206,47.409,159.366
C06828=1027.859,361.894,360.786,172.200,47.408,159.365
C06829=1027.851,361.648,360.825,172.192,47.407,159.364
C06830=1027.843,361.400,360.864,172.185,47.406,159.363
C06831=1027.836,361.154,360.903,172.177,47.405,159.362
C06832=1027.827,360.907,360.942,172.171,47.404,159.361
C06833=1027.819,360.660,360.981,172.164,47.403,159.359
C06834=1027.811,360.413,361.020,172.156,47.402,159.358
C06835=1027.803,360.167,361.058,172.149,47.401,159.357
C06836=1027.795,359.920,361.097,172.143,47.400,159.356
C06837=1027.787,359.673,361.136,172.135,47.400,159.355
C06838=1027.779,359.426,361.175,172.128,47.398,159.353
C06839=1027.771,359.180,361.214,172.120,47.397,159.352
C06840=1027.763,358.932,361.252,172.114,47.396,159.351
C06841=1027.754,358.685,361.291,172.107,47.396,159.350
C06842=1027.747,358.439,361.329,172.099,47.395,159.349
C06843=1027.739,358.192,361.368,172.092,47.394,159.348
C06844=1027.731,357.944,361.406,172.086,47.393,159.347
C06845=1027.723,357.698,361.445,172.078,47.392,159.345
C06846=1027.715,357.451,361.483,172.071,47.391,159.344
C06847=1027.707,357.203,361.522,172.065,47.390,159.343
C06848=1027.699,356.957,361.560,172.057,47.389,159.342
C06849=1027.691,356.710,361.599,172.050,47.389,159.341
C06850=1027.683,356.463,361.637,172.044,47.388,159.340
C06851=1027.675,356.216,361.675,172.037,47.388,159.339
C06852=1027.667,355.970,361.713,172.029,47.387,159.338
C06853=1027.659,355.722,361.752,172.023,47.386,159.337
C06854=1027.651,355.475,361.790,172.016,47.385,159.336
C06855=1027.643,355.229,361.829,172.009,47.384,159.334
C06856=1027.635,354.982,361.867,172.002,47.383,159.333
C06857=1027.628,354.734,361.905,171.995,47.383,159.332
C06858=1027.620,354.487,361.943,171.989,47.382,159.331
C06859=1027.611,354.241,361.981,171.982,47.382,159.330
C06860=1027.604,353.994,362.019,171.974,47.381,159.329
C06861=1027.596,353.747,362.057,171.968,47.380,159.328
C06862=1027.588,353.500,362.095,171.961,47.380,159.327
C06863=1027.580,353.253,362.133,171.955,47.379,159.326
C06864=1027.572,353.006,362.171,171.948,47.378,159.325
C06865=1027.564,352.758,362.209,171.941,47.378,159.324
C06866=1027.556,352.512,362.246,171.934,47.377,159.323
C06867=1027.549,352.265,362.284,171.927,47.377,159.322
C06868=1027.541,352.018,362.323,171.921,47.376,159.321
C06869=1027.533,351.771,362.360,171.914,47.375,159.320
C06870=1027.526,351.554,362.393,171.908,47.375,159.319
C06871=1027.519,351.336,362.426,171.902,47.374,159.318
C06872=1027.513,351.119,362.460,171.897,47.373,159.317
C06873=1027.506,350.901,362.493,171.891,47.373,159.316
C06874=1027.499,350.684,362.526,171.885,47.372,159.315
C06875=1027.492,350.466,362.560,171.879,47.372,159.314
C06876=1027.485,350.249,362.592,171.873,47.372,159.314
C06877=1027.478,350.032,362.626,171.867,47.371,159.313
C06878=1027.471,349.785,362.663,171.861,47.371,159.312
C06879=1027.464,349.538,362.701,171.854,47.370,159.311
C06880=1027.455,349.291,362.739,171.848,47.370,159.310
C06881=1027.447,349.044,362.776,171.841,47.370,159.309
C06882=1027.440,348.796,362.814,171.834,47.368,159.308
C06883=1027.432,348.550,362.851,171.827,47.368,159.307
C06884=1027.425,348.303,362.888,171.821,47.368,159.306
C06885=1027.417,348.055,362.926,171.815,47.367,159.305
C06886=1027.409,347.808,362.963,171.808,47.367,159.304
C06887=1027.402,347.561,363.001,171.802,47.366,159.303
C06888=1027.394,347.314,363.037,171.795,47.366,159.302
C06889=1027.386,347.067,363.074,171.789,47.366,159.301
C06890=1027.379,346.820,363.112,171.782,47.366,159.300
C06891=1027.370,346.572,363.149,171.776,47.365,159.299
C06892=1027.363,346.325,363.187,171.769,47.365,159.298
C06893=1027.355,346.078,363.224,171.763,47.365,159.297
C06894=1027.348,345.831,363.261,171.757,47.364,159.297
C06895=1027.340,345.584,363.297,171.750,47.364,159.296
C06896=1027.333,345.337,363.335,171.744,47.364,159.295
C06897=1027.325,345.090,363.372,171.737,47.363,159.294
C06898=1027.318,344.843,363.409,171.731,47.363,159.293
C06899=1027.310,344.595,363.446,171.725,47.363,159.292
C06900=1027.302,344.348,363.483,171.718,47.362,159.291
C06901=1027.295,344.101,363.520,171.712,47.362,159.290
C06902=1027.287,343.854,363.556,171.705,47.362,159.289
C06903=1027.280,343.607,363.594,171.699,47.361,159.288
C06904=1027.272,343.360,363.631,171.693,47.361,159.288
C06905=1027.264,343.113,363.667,171.686,47.361,159.287
C06906=1027.257,342.865,363.705,171.681,47.361,159.286
C06907=1027.249,342.618,363.741,171.675,47.361,159.285
C06908=1027.242,342.371,363.778,171.668,47.361,159.284
C06909=1027.234,342.123,363.814,171.662,47.360,159.283
C06910=1027.226,341.877,363.851,171.656,47.360,159.282
C06911=1027.219,341.629,363.888,171.649,47.360,159.282
C06912=1027.212,341.383,363.925,171.643,47.360,159.281
C06913=1027.204,341.135,363.961,171.637,47.359,159.280
C06914=1027.197,340.887,363.998,171.631,47.360,159.279
C06915=1027.189,340.641,364.035,171.625,47.359,159.278
C06916=1027.182,340.393,364.071,171.619,47.359,159.277
C06917=1027.175,340.145,364.108,171.613,47.359,159.277
C06918=1027.167,339.899,364.144,171.606,47.359,159.276
C06919=1027.160,339.652,364.181,171.600,47.359,159.275
C06920=1027.152,339.404,364.217,171.594,47.359,159.274
C06921=1027.144,339.157,364.253,171.587,47.358,159.273
C06922=1027.137,338.910,364.289,171.582,47.359,159.272
C06923=1027.129,338.663,364.326,171.576,47.359,159.272
C06924=1027.122,338.416,364.362,171.569,47.359,159.271
C06925=1027.114,338.168,364.398,171.563,47.359,159.270
C06926=1027.107,337.921,364.435,171.557,47.358,159.269
C06927=1027.099,337.673,364.471,171.552,47.359,159.268
C06928=1027.092,337.427,364.507,171.545,47.358,159.267
C06929=1027.085,337.179,364.543,171.539,47.359,159.267
C06930=1027.078,336.960,364.575,171.534,47.358,159.266
C06931=1027.071,336.741,364.607,171.529,47.359,159.265
C06932=1027.065,336.522,364.639,171.523,47.359,159.265
C06933=1027.058,336.303,364.671,171.519,47.359,159.264
C06934=1027.052,336.085,364.702,171.513,47.359,159.263
C06935=1027.045,335.865,364.735,171.507,47.359,159.263
C06936=1027.039,335.646,364.767,171.503,47.359,159.262
C06937=1027.032,335.428,364.799,171.497,47.359,159.261
C06938=1027.025,335.180,364.834,171.491,47.359,159.260
C06939=1027.017,334.933,364.870,171.485,47.359,159.260
C06940=1027.010,334.685,364.907,171.480,47.359,159.259
C06941=1027.003,334.438,364.943,171.473,47.359,159.258
C06942=1026.996,334.191,364.979,171.467,47.359,159.257
C06943=1026.989,333.943,365.014,171.461,47.359,159.257
C06944=1026.981,333.696,365.050,171.456,47.359,159.256
C06945=1026.974,333.449,365.086,171.450,47.360,159.255
C06946=1026.966,333.202,365.121,171.443,47.360,159.255
C06947=1026.958,332.954,365.157,171.438,47.360,159.254
C06948=1026.952,332.707,365.193,171.432,47.360,159.253
C06949=1026.944,332.459,365.229,171.426,47.361,159.252
C06950=1026.937,332.213,365.265,171.421,47.361,159.252
C06951=1026.929,331.964,365.300,171.415,47.361,159.251
C06952=1026.922,331.718,365.335,171.408,47.361,159.250
C06953=1026.914,331.470,365.371,171.403,47.361,159.250
C06954=1026.907,331.223,365.406,171.397,47.362,159.249
C06955=1026.900,330.975,365.442,171.391,47.362,159.248
C06956=1026.893,330.728,365.477,171.386,47.362,159.248
C06957=1026.885,330.480,365.514,171.380,47.362,159.247
C06958=1026.878,330.233,365.548,171.374,47.362,159.246
C06959=1026.871,329.986,365.583,171.368,47.363,159.246
C06960=1026.863,329.738,365.619,171.362,47.364,159.245
C06961=1026.857,329.491,365.655,171.357,47.364,159.244
C06962=1026.849,329.243,365.690,171.351,47.364,159.243
C06963=1026.842,328.996,365.726,171.345,47.364,159.243
C06964=1026.835,328.749,365.760,171.340,47.364,159.242
C06965=1026.827,328.501,365.796,171.334,47.365,159.242
C06966=1026.821,328.254,365.831,171.329,47.365,159.241
C06967=1026.813,328.007,365.867,171.323,47.365,159.240
C06968=1026.806,327.759,365.902,171.317,47.366,159.239
C06969=1026.799,327.512,365.937,171.312,47.366,159.239
C06970=1026.792,327.265,365.972,171.305,47.367,159.238
C06971=1026.784,327.017,366.007,171.300,47.367,159.237
C06972=1026.777,326.769,366.042,171.294,47.368,159.237
C06973=1026.769,326.522,366.077,171.289,47.368,159.236
C06974=1026.762,326.274,366.112,171.283,47.369,159.236
C06975=1026.755,326.027,366.147,171.278,47.369,159.235
C06976=1026.747,325.780,366.181,171.272,47.370,159.235
C06977=1026.740,325.532,366.216,171.267,47.370,159.234
C06978=1026.732,325.284,366.251,171.261,47.371,159.233
C06979=1026.725,325.037,366.285,171.255,47.371,159.233
C06980=1026.718,324.790,366.320,171.249,47.372,159.232
C06981=1026.710,324.542,366.355,171.244,47.373,159.232
C06982=1026.704,324.294,366.390,171.238,47.373,159.231
C06983=1026.696,324.047,366.424,171.233,47.374,159.230
C06984=1026.689,323.800,366.459,171.227,47.374,159.230
C06985=1026.682,323.553,366.494,171.222,47.375,159.229
C06986=1026.674,323.304,366.528,171.216,47.375,159.229
C06987=1026.667,323.057,366.563,171.211,47.375,159.228
C06988=1026.660,322.810,366.598,171.205,47.376,159.227
C06989=1026.653,322.562,366.632,171.200,47.377,159.227
C06990=1026.646,322.341,366.663,171.194,47.377,159.226
C06991=1026.640,322.120,366.694,171.190,47.378,159.226
C06992=1026.634,321.899,366.725,171.185,47.378,159.225
C06993=1026.627,321.677,366.755,171.180,47.379,159.225
C06994=1026.620,321.457,366.786,171.175,47.380,159.224
C06995=1026.614,321.235,366.817,171.171,47.380,159.224
C06996=1026.608,321.014,366.848,171.165,47.381,159.223
C06997=1026.601,320.793,366.879,171.161,47.382,159.223
C06998=1026.594,320.545,366.913,171.155,47.382,159.222
C06999=1026.587,320.298,366.947,171.150,47.383,159.222
C07000=1026.580,320.050,366.982,171.145,47.383,159.221
C07001=1026.573,319.803,367.016,171.139,47.384,159.221
C07002=1026.565,319.556,367.051,171.134,47.385,159.220
C07003=1026.559,319.308,367.085,171.128,47.385,159.219
C07004=1026.551,319.061,367.120,171.123,47.386,159.219
C07005=1026.545,318.813,367.154,171.118,47.387,159.218
C07006=1026.538,318.565,367.188,171.112,47.387,159.218
C07007=1026.530,318.318,367.222,171.107,47.388,159.217
C07008=1026.524,318.070,367.257,171.102,47.389,159.217
C07009=1026.516,317.822,367.291,171.096,47.390,159.216
C07010=1026.509,317.575,367.325,171.091,47.391,159.216
C07011=1026.502,317.327,367.360,171.085,47.391,159.215
C07012=1026.495,317.080,367.393,171.081,47.392,159.215
C07013=1026.488,316.833,367.428,171.076,47.393,159.214
C07014=1026.482,316.585,367.462,171.070,47.393,159.214
C07015=1026.475,316.338,367.496,171.065,47.394,159.213
C07016=1026.467,316.090,367.530,171.060,47.395,159.213
C07017=1026.461,315.842,367.564,171.054,47.396,159.212
C07018=1026.453,315.595,367.599,171.049,47.396,159.212
C07019=1026.446,315.347,367.632,171.044,47.397,159.211
C07020=1026.440,315.100,367.666,171.038,47.398,159.211
C07021=1026.433,314.852,367.700,171.033,47.399,159.210
C07022=1026.426,314.605,367.734,171.028,47.400,159.210
C07023=1026.419,314.357,367.768,171.023,47.400,159.209
C07024=1026.412,314.109,367.802,171.018,47.401,159.209
C07025=1026.406,313.862,367.836,171.013,47.402,159.208
C07026=1026.398,313.615,367.870,171.007,47.402,159.208
C07027=1026.392,313.367,367.905,171.002,47.404,159.207
C07028=1026.385,313.119,367.939,170.997,47.405,159.207
C07029=1026.378,312.872,367.972,170.991,47.405,159.206
C07030=1026.372,312.624,368.006,170.987,47.406,159.206
C07031=1026.364,312.377,368.040,170.982,47.407,159.205
C07032=1026.358,312.130,368.074,170.976,47.407,159.205
C07033=1026.351,311.882,368.108,170.971,47.409,159.204
C07034=1026.344,311.633,368.141,170.966,47.410,159.204
C07035=1026.338,311.386,368.175,170.961,47.410,159.203
C07036=1026.331,311.139,368.209,170.955,47.411,159.203
C07037=1026.324,310.891,368.243,170.951,47.412,159.203
C07038=1026.317,310.644,368.276,170.946,47.413,159.202
C07039=1026.310,310.396,368.310,170.941,47.414,159.201
C07040=1026.303,310.148,368.343,170.935,47.415,159.201
C07041=1026.296,309.901,368.376,170.930,47.417,159.201
C07042=1026.289,309.653,368.409,170.925,47.418,159.200
C07043=1026.281,309.405,368.443,170.920,47.419,159.200
C07044=1026.275,309.158,368.476,170.915,47.420,159.199
C07045=1026.268,308.910,368.509,170.911,47.421,159.199
C07046=1026.260,308.663,368.542,170.905,47.422,159.199
C07047=1026.254,308.415,368.575,170.900,47.423,159.198
C07048=1026.246,308.168,368.609,170.895,47.424,159.198
C07049=1026.239,307.920,368.641,170.890,47.425,159.197
C07050=1026.233,307.701,368.671,170.886,47.426,159.197
C07051=1026.227,307.482,368.700,170.880,47.427,159.197
C07052=1026.220,307.264,368.729,170.876,47.428,159.196
C07053=1026.215,307.045,368.758,170.872,47.429,159.196
C07054=1026.208,306.826,368.788,170.868,47.431,159.196
C07055=1026.203,306.607,368.817,170.863,47.431,159.195
C07056=1026.196,306.389,368.846,170.859,47.432,159.195
C07057=1026.190,306.170,368.875,170.855,47.434,159.195
C07058=1026.183,305.922,368.908,170.850,47.434,159.194
C07059=1026.176,305.675,368.941,170.845,47.436,159.194
C07060=1026.169,305.427,368.974,170.840,47.437,159.194
C07061=1026.162,305.180,369.007,170.835,47.439,159.193
C07062=1026.155,304.932,369.040,170.830,47.439,159.193
C07063=1026.148,304.684,369.072,170.825,47.440,159.192
C07064=1026.141,304.436,369.105,170.820,47.442,159.192
C07065=1026.135,304.189,369.139,170.815,47.443,159.192
C07066=1026.127,303.941,369.171,170.810,47.444,159.191
C07067=1026.121,303.693,369.204,170.805,47.445,159.191
C07068=1026.114,303.445,369.237,170.801,47.447,159.191
C07069=1026.107,303.198,369.269,170.796,47.448,159.190
C07070=1026.100,302.951,369.303,170.791,47.449,159.190
C07071=1026.093,302.703,369.336,170.785,47.451,159.190
C07072=1026.086,302.455,369.368,170.780,47.452,159.189
C07073=1026.079,302.207,369.401,170.776,47.453,159.189
C07074=1026.073,301.959,369.434,170.771,47.454,159.189
C07075=1026.066,301.712,369.466,170.766,47.456,159.188
C07076=1026.059,301.464,369.499,170.761,47.457,159.188
C07077=1026.052,301.217,369.531,170.757,47.458,159.188
C07078=1026.045,300.968,369.565,170.752,47.460,159.187
C07079=1026.039,300.721,369.597,170.747,47.461,159.187
C07080=1026.032,300.473,369.629,170.742,47.462,159.187
C07081=1026.025,300.225,369.663,170.738,47.463,159.186
C07082=1026.019,299.977,369.695,170.733,47.465,159.186
C07083=1026.012,299.730,369.727,170.728,47.466,159.186
C07084=1026.005,299.482,369.761,170.723,47.468,159.185
C07085=1025.999,299.234,369.793,170.719,47.469,159.185
C07086=1025.992,298.987,369.825,170.714,47.470,159.185
C07087=1025.985,298.739,369.858,170.709,47.472,159.184
C07088=1025.978,298.491,369.891,170.703,47.473,159.184
C07089=1025.971,298.244,369.923,170.699,47.474,159.184
C07090=1025.965,297.996,369.955,170.694,47.476,159.183
C07091=1025.959,297.748,369.988,170.689,47.477,159.183
C07092=1025.951,297.500,370.021,170.685,47.478,159.183
C07093=1025.945,297.252,370.053,170.680,47.480,159.182
C07094=1025.939,297.005,370.086,170.675,47.481,159.182
C07095=1025.932,296.757,370.118,170.670,47.482,159.182
C07096=1025.926,296.509,370.150,170.666,47.484,159.181
C07097=1025.918,296.261,370.183,170.661,47.485,159.181
C07098=1025.912,296.014,370.216,170.656,47.486,159.181
C07099=1025.906,295.766,370.248,170.652,47.488,159.181
C07100=1025.899,295.518,370.280,170.647,47.490,159.180
C07101=1025.893,295.271,370.313,170.642,47.491,159.180
C07102=1025.887,295.022,370.345,170.638,47.492,159.180
C07103=1025.879,294.774,370.377,170.633,47.493,159.179
C07104=1025.873,294.527,370.410,170.628,47.495,159.179
C07105=1025.866,294.279,370.441,170.624,47.497,159.179
C07106=1025.860,294.031,370.474,170.619,47.498,159.179
C07107=1025.853,293.784,370.505,170.614,47.499,159.178
C07108=1025.847,293.536,370.538,170.610,47.501,159.178
C07109=1025.840,293.288,370.570,170.606,47.503,159.178
C07110=1025.834,293.078,370.597,170.602,47.504,159.178
C07111=1025.828,292.868,370.624,170.598,47.505,159.177
C07112=1025.823,292.657,370.651,170.594,47.507,159.177
C07113=1025.817,292.448,370.679,170.590,47.508,159.177
C07114=1025.811,292.237,370.706,170.586,47.509,159.177
C07115=1025.805,292.028,370.732,170.582,47.511,159.176
C07116=1025.800,291.817,370.759,170.578,47.512,159.176
C07117=1025.794,291.608,370.787,170.574,47.514,159.176
C07118=1025.787,291.360,370.818,170.569,47.515,159.176
C07119=1025.781,291.112,370.850,170.565,47.517,159.176
C07120=1025.774,290.864,370.881,170.560,47.518,159.175
C07121=1025.767,290.617,370.913,170.556,47.520,159.175
C07122=1025.760,290.369,370.945,170.552,47.521,159.175
C07123=1025.754,290.121,370.977,170.547,47.523,159.175
C07124=1025.747,289.872,371.008,170.542,47.525,159.174
C07125=1025.740,289.625,371.041,170.538,47.527,159.174
C07126=1025.733,289.377,371.072,170.533,47.528,159.174
C07127=1025.726,289.129,371.104,170.528,47.530,159.174
C07128=1025.720,288.881,371.135,170.524,47.531,159.174
C07129=1025.714,288.633,371.167,170.520,47.533,159.173
C07130=1025.707,288.385,371.198,170.515,47.535,159.173
C07131=1025.700,288.137,371.230,170.511,47.536,159.173
C07132=1025.694,287.889,371.261,170.506,47.539,159.173
C07133=1025.687,287.641,371.293,170.501,47.541,159.173
C07134=1025.680,287.393,371.324,170.497,47.542,159.172
C07135=1025.673,287.145,371.356,170.493,47.544,159.172
C07136=1025.667,286.897,371.387,170.488,47.546,159.172
C07137=1025.661,286.650,371.418,170.484,47.547,159.172
C07138=1025.654,286.402,371.449,170.479,47.549,159.172
C07139=1025.647,286.154,371.481,170.474,47.551,159.171
C07140=1025.641,285.906,371.513,170.470,47.552,159.171
C07141=1025.634,285.658,371.544,170.466,47.554,159.171
C07142=1025.628,285.410,371.576,170.461,47.556,159.171
C07143=1025.620,285.163,371.607,170.457,47.558,159.171
C07144=1025.614,284.915,371.638,170.452,47.560,159.171
C07145=1025.607,284.667,371.670,170.447,47.562,159.170
C07146=1025.600,284.418,371.700,170.444,47.563,159.170
C07147=1025.594,284.171,371.732,170.439,47.565,159.170
C07148=1025.587,283.923,371.763,170.434,47.567,159.170
C07149=1025.580,283.675,371.795,170.431,47.569,159.170
C07150=1025.574,283.427,371.824,170.426,47.571,159.169
C07151=1025.567,283.179,371.856,170.421,47.573,159.169
C07152=1025.560,282.931,371.887,170.417,47.575,159.169
C07153=1025.554,282.683,371.918,170.413,47.577,159.169
C07154=1025.547,282.435,371.949,170.409,47.578,159.169
C07155=1025.540,282.187,371.981,170.404,47.580,159.169
C07156=1025.533,281.939,372.011,170.399,47.582,159.168
C07157=1025.527,281.692,372.042,170.395,47.584,159.168
C07158=1025.520,281.444,372.073,170.391,47.586,159.168
C07159=1025.514,281.195,372.104,170.386,47.588,159.168
C07160=1025.507,280.947,372.136,170.382,47.590,159.168
C07161=1025.501,280.699,372.166,170.378,47.592,159.168
C07162=1025.495,280.452,372.197,170.374,47.594,159.168
C07163=1025.487,280.204,372.228,170.369,47.596,159.167
C07164=1025.481,279.956,372.259,170.364,47.598,159.167
C07165=1025.474,279.708,372.290,170.361,47.600,159.167
C07166=1025.468,279.459,372.321,170.356,47.602,159.167
C07167=1025.461,279.212,372.352,170.352,47.604,159.167
C07168=1025.455,278.963,372.383,170.347,47.606,159.167
C07169=1025.448,278.716,372.414,170.343,47.608,159.167
C07170=1025.437,278.308,372.464,170.336,47.611,159.166
C07171=1025.427,277.900,372.515,170.329,47.615,159.166
C07172=1025.416,277.492,372.566,170.322,47.618,159.166
C07173=1025.405,277.084,372.616,170.315,47.621,159.166
C07174=1025.399,276.836,372.647,170.311,47.623,159.166
C07175=1025.392,276.588,372.678,170.306,47.625,159.166
C07176=1025.385,276.340,372.708,170.302,47.627,159.166
C07177=1025.379,276.092,372.739,170.298,47.630,159.166
C07178=1025.372,275.843,372.769,170.294,47.632,159.165
C07179=1025.366,275.596,372.800,170.290,47.634,159.165
C07180=1025.359,275.348,372.830,170.286,47.636,159.165
C07181=1025.352,275.100,372.861,170.281,47.638,159.165
C07182=1025.346,274.852,372.891,170.277,47.640,159.165
C07183=1025.339,274.604,372.921,170.272,47.642,159.165
C07184=1025.333,274.356,372.951,170.269,47.645,159.165
C07185=1025.326,274.108,372.982,170.264,47.647,159.165
C07186=1025.319,273.860,373.013,170.259,47.649,159.165
C07187=1025.314,273.612,373.043,170.256,47.651,159.165
C07188=1025.306,273.364,373.073,170.251,47.653,159.165
C07189=1025.300,273.115,373.104,170.248,47.655,159.164
C07190=1025.293,272.868,373.134,170.243,47.658,159.164
C07191=1025.287,272.619,373.165,170.239,47.659,159.164
C07192=1025.280,272.371,373.194,170.235,47.662,159.164
C07193=1025.274,272.123,373.225,170.230,47.664,159.164
C07194=1025.267,271.875,373.255,170.227,47.666,159.164
C07195=1025.261,271.627,373.286,170.222,47.669,159.164
C07196=1025.254,271.379,373.316,170.218,47.670,159.164
C07197=1025.248,271.131,373.346,170.214,47.673,159.164
C07198=1025.241,270.883,373.376,170.209,47.675,159.164
C07199=1025.235,270.635,373.406,170.206,47.678,159.164
C07200=1025.228,270.387,373.437,170.201,47.680,159.164
C07201=1025.222,270.139,373.467,170.198,47.682,159.164
C07202=1025.215,269.891,373.497,170.193,47.684,159.164
C07203=1025.208,269.643,373.527,170.190,47.687,159.164
C07204=1025.202,269.394,373.557,170.185,47.689,159.164
C07205=1025.196,269.146,373.587,170.182,47.691,159.164
C07206=1025.189,268.898,373.617,170.177,47.693,159.163
C07207=1025.183,268.650,373.647,170.172,47.696,159.163
C07208=1025.176,268.402,373.677,170.169,47.698,159.164
C07209=1025.169,268.154,373.706,170.164,47.700,159.163
C07210=1025.163,267.906,373.737,170.161,47.703,159.163
C07211=1025.156,267.658,373.767,170.156,47.705,159.163
C07212=1025.150,267.409,373.796,170.153,47.707,159.163
C07213=1025.144,267.161,373.826,170.148,47.710,159.163
C07214=1025.137,266.913,373.857,170.144,47.712,159.163
C07215=1025.130,266.666,373.886,170.140,47.715,159.163
C07216=1025.124,266.417,373.916,170.136,47.717,159.163
C07217=1025.117,266.169,373.946,170.132,47.719,159.163
C07218=1025.110,265.920,373.975,170.128,47.722,159.163
C07219=1025.104,265.673,374.005,170.124,47.724,159.163
C07220=1025.097,265.425,374.035,170.120,47.727,159.163
C07221=1025.091,265.176,374.065,170.116,47.729,159.163
C07222=1025.085,264.928,374.095,170.112,47.731,159.163
C07223=1025.078,264.680,374.124,170.107,47.734,159.163
C07224=1025.071,264.432,374.154,170.104,47.737,159.163
C07225=1025.064,264.183,374.183,170.099,47.739,159.163
C07226=1025.054,263.780,374.232,170.093,47.743,159.163
C07227=1025.044,263.378,374.280,170.087,47.747,159.163
C07228=1025.034,262.974,374.328,170.080,47.751,159.163
C07229=1025.023,262.571,374.376,170.074,47.755,159.163
C07230=1025.016,262.322,374.405,170.069,47.757,159.163
C07231=1025.010,262.075,374.435,170.066,47.760,159.163
C07232=1025.003,261.827,374.464,170.061,47.763,159.163
C07233=1024.996,261.578,374.494,170.058,47.765,159.163
C07234=1024.991,261.330,374.524,170.054,47.768,159.163
C07235=1024.984,261.082,374.553,170.050,47.770,159.163
C07236=1024.977,260.834,374.583,170.046,47.773,159.163
C07237=1024.971,260.586,374.612,170.042,47.775,159.164
C07238=1024.965,260.337,374.641,170.038,47.778,159.164
C07239=1024.957,260.089,374.670,170.034,47.781,159.164
C07240=1024.951,259.841,374.699,170.030,47.783,159.164
C07241=1024.945,259.593,374.728,170.026,47.786,159.164
C07242=1024.937,259.344,374.758,170.022,47.788,159.164
C07243=1024.930,259.097,374.787,170.018,47.791,159.164
C07244=1024.924,258.848,374.816,170.014,47.794,159.164
C07245=1024.917,258.600,374.845,170.010,47.796,159.164
C07246=1024.911,258.351,374.874,170.006,47.800,159.164
C07247=1024.904,258.104,374.903,170.003,47.802,159.164
C07248=1024.897,257.855,374.932,169.998,47.805,159.164
C07249=1024.891,257.607,374.961,169.994,47.807,159.164
C07250=1024.885,257.359,374.990,169.990,47.810,159.164
C07251=1024.878,257.111,375.019,169.986,47.813,159.164
C07252=1024.871,256.862,375.048,169.983,47.816,159.164
C07253=1024.865,256.614,375.077,169.979,47.818,159.164
C07254=1024.858,256.366,375.106,169.975,47.821,159.164
C07255=1024.851,256.118,375.135,169.971,47.824,159.164
C07256=1024.845,255.869,375.164,169.967,47.826,159.165
C07257=1024.838,255.621,375.193,169.963,47.829,159.165
C07258=1024.832,255.373,375.222,169.959,47.832,159.165
C07259=1024.825,255.125,375.250,169.955,47.835,159.165
C07260=1024.818,254.876,375.280,169.951,47.837,159.165
C07261=1024.812,254.628,375.309,169.948,47.840,159.165
C07262=1024.806,254.379,375.337,169.944,47.843,159.165
C07263=1024.799,254.131,375.366,169.940,47.846,159.165
C07264=1024.793,253.883,375.395,169.936,47.848,159.165
C07265=1024.787,253.635,375.424,169.933,47.851,159.165
C07266=1024.779,253.387,375.453,169.928,47.854,159.165
C07267=1024.773,253.138,375.482,169.925,47.857,159.165
C07268=1024.767,252.890,375.511,169.921,47.860,159.166
C07269=1024.761,252.642,375.539,169.916,47.863,159.166
C07270=1024.754,252.394,375.567,169.913,47.865,159.166
C07271=1024.747,252.146,375.596,169.909,47.869,159.166
C07272=1024.741,251.897,375.625,169.906,47.871,159.166
C07273=1024.734,251.649,375.655,169.901,47.874,159.166
C07274=1024.728,251.400,375.683,169.898,47.877,159.166
C07275=1024.721,251.152,375.712,169.894,47.880,159.166
C07276=1024.715,250.904,375.741,169.890,47.882,159.166
C07277=1024.708,250.656,375.769,169.886,47.885,159.166
C07278=1024.702,250.407,375.797,169.883,47.888,159.167
C07279=1024.696,250.159,375.827,169.878,47.891,159.167
C07280=1024.690,249.911,375.856,169.875,47.894,159.167
